(* IEC 61131-3 sources: TIA2AX/tests/V18/test_projects/expected/HW_2200330/ST60_PLC, 7 files *)

(* ---- HwIdentifiers.st ---- *)
TYPE
	HwIdentifiers : WORD
	(
		ST60_PLC_Profilschiene_0 :=	WORD#256,
		ST60_PLC :=	WORD#48,
		ST60_PLC_Card_reader_writer_1 :=	WORD#51,
		ST60_PLC_CPU_display_1 :=	WORD#54,
		ST60_PLC_OPC_UA_1 :=	WORD#117,
		ST60_PLC_DP_interface_1 :=	WORD#60,
		ST60_PLC_PROFINET_interface_1 :=	WORD#64,
		ST60_PLC_PROFINET_interface_1_Port_1 :=	WORD#65,
		ST60_PLC_PROFINET_interface_1_Port_2 :=	WORD#66,
		ST60_PLC_PROFINET_interface_2 :=	WORD#72,
		ST60_PLC_PROFINET_interface_2_Port_1 :=	WORD#73,
		ST60_Switch_SCALANCE_X_rack :=	WORD#421,
		ST60_Switch :=	WORD#422,
		ST60_Switch_ST60_Switch :=	WORD#423,
		ST60_Switch_SCALANCE_interface_1 :=	WORD#424,
		ST60_Switch_SCALANCE_interface_1_Port_1 :=	WORD#425,
		ST60_Switch_SCALANCE_interface_1_Port_2 :=	WORD#426,
		ST60_Switch_SCALANCE_interface_1_Port_3 :=	WORD#427,
		ST60_Switch_SCALANCE_interface_1_Port_4 :=	WORD#428,
		ST60_Switch_SCALANCE_interface_1_Port_5 :=	WORD#429,
		ST60_Switch_SCALANCE_interface_1_Port_6 :=	WORD#430,
		ST60_Switch_SCALANCE_interface_1_Port_7 :=	WORD#431,
		ST60_Switch_SCALANCE_interface_1_Port_8 :=	WORD#432,
		ST60_Switch_SCALANCE_interface_1_Port_9 :=	WORD#433,
		ST60_Switch_SCALANCE_interface_1_Port_10 :=	WORD#434,
		ST60_Switch_SCALANCE_interface_1_Port_11 :=	WORD#435,
		ST60_Switch_SCALANCE_interface_1_Port_12 :=	WORD#436,
		ST60_Switch_SCALANCE_interface_1_Port_13 :=	WORD#437,
		ST60_Switch_SCALANCE_interface_1_Port_14 :=	WORD#438,
		ST60_Switch_SCALANCE_interface_1_Port_15 :=	WORD#439,
		ST60_Switch_SCALANCE_interface_1_Port_16 :=	WORD#440,
		ST60_Switch_1_SCALANCE_X_rack :=	WORD#445,
		ST60_Switch_1 :=	WORD#446,
		ST60_Switch_1_ST60_Switch_1 :=	WORD#447,
		ST60_Switch_1_SCALANCE_interface_1 :=	WORD#448,
		ST60_Switch_1_SCALANCE_interface_1_Port_1 :=	WORD#449,
		ST60_Switch_1_SCALANCE_interface_1_Port_2 :=	WORD#450,
		ST60_Switch_1_SCALANCE_interface_1_Port_3 :=	WORD#451,
		ST60_Switch_1_SCALANCE_interface_1_Port_4 :=	WORD#452,
		ST60_Switch_1_SCALANCE_interface_1_Port_5 :=	WORD#453,
		ST60_Switch_1_SCALANCE_interface_1_Port_6 :=	WORD#454,
		ST60_Switch_1_SCALANCE_interface_1_Port_7 :=	WORD#455,
		ST60_Switch_1_SCALANCE_interface_1_Port_8 :=	WORD#456,
		ST60_Switch_1_SCALANCE_interface_1_Port_9 :=	WORD#457,
		ST60_Switch_1_SCALANCE_interface_1_Port_10 :=	WORD#458,
		ST60_Switch_1_SCALANCE_interface_1_Port_11 :=	WORD#459,
		ST60_Switch_1_SCALANCE_interface_1_Port_12 :=	WORD#460,
		ST60_Switch_1_SCALANCE_interface_1_Port_13 :=	WORD#461,
		ST60_Switch_1_SCALANCE_interface_1_Port_14 :=	WORD#462,
		ST60_Switch_1_SCALANCE_interface_1_Port_15 :=	WORD#463,
		ST60_Switch_1_SCALANCE_interface_1_Port_16 :=	WORD#464,
		ST60_2_DM260_Rack :=	WORD#270,
		ST60_2_DM260 :=	WORD#258,
		ST60_2_DM260_Interface :=	WORD#259,
		ST60_2_DM260_Interface_Port_1 :=	WORD#260,
		ST60_2_DM260_DataMan_260 :=	WORD#261,
		ST60_2_DM260_Acquisition_Control :=	WORD#262,
		ST60_2_DM260_Acquisition_Status :=	WORD#263,
		ST60_2_DM260_Results_Control :=	WORD#264,
		ST60_2_DM260_Results_Status :=	WORD#265,
		ST60_2_DM260_Soft_Event_Control :=	WORD#266,
		ST60_2_DM260_User_Data_64_bytes :=	WORD#267,
		ST60_2_DM260_Result_Data_64_bytes :=	WORD#268,
		ST60_1_DM260_Rack :=	WORD#272,
		ST60_1_DM260 :=	WORD#273,
		ST60_1_DM260_Interface :=	WORD#274,
		ST60_1_DM260_Interface_Port_1 :=	WORD#275,
		ST60_1_DM260_DataMan_260 :=	WORD#276,
		ST60_1_DM260_Acquisition_Control :=	WORD#277,
		ST60_1_DM260_Acquisition_Status :=	WORD#278,
		ST60_1_DM260_Results_Control :=	WORD#279,
		ST60_1_DM260_Results_Status :=	WORD#280,
		ST60_1_DM260_Soft_Event_Control :=	WORD#281,
		ST60_1_DM260_User_Data_64_bytes :=	WORD#282,
		ST60_1_DM260_Result_Data_64_bytes :=	WORD#283,
		ST60_1_DM260_WPC_Rack :=	WORD#285,
		ST60_1_DM260_WPC :=	WORD#286,
		ST60_1_DM260_WPC_Interface :=	WORD#287,
		ST60_1_DM260_WPC_Interface_Port_1 :=	WORD#288,
		ST60_1_DM260_WPC_DataMan_260 :=	WORD#289,
		ST60_1_DM260_WPC_Acquisition_Control :=	WORD#290,
		ST60_1_DM260_WPC_Acquisition_Status :=	WORD#291,
		ST60_1_DM260_WPC_Results_Control :=	WORD#292,
		ST60_1_DM260_WPC_Results_Status :=	WORD#293,
		ST60_1_DM260_WPC_Soft_Event_Control :=	WORD#294,
		ST60_1_DM260_WPC_User_Data_64_bytes :=	WORD#295,
		ST60_1_DM260_WPC_Result_Data_64_bytes :=	WORD#296,
		ST60_TZ535_PN_Rack :=	WORD#298,
		ST60_TZ535_PN :=	WORD#299,
		ST60_TZ535_PN_Interface :=	WORD#300,
		ST60_TZ535_PN_Interface_Port_1 :=	WORD#301,
		ST60_TZ535_PN_Interface_Port_2 :=	WORD#302,
		ST60_TZ535_PN_2D_TZ535_PN_PROFINET_IO :=	WORD#303,
		ST60_TZ535_PN_In_Out_32_byte_x :=	WORD#304,
		ST60_SCHUNK_R_Rack :=	WORD#306,
		ST60_SCHUNK_R :=	WORD#307,
		ST60_SCHUNK_R_Interface :=	WORD#308,
		ST60_SCHUNK_R_Interface_Port_1 :=	WORD#309,
		ST60_SCHUNK_R_Interface_Port_2 :=	WORD#310,
		ST60_SCHUNK_R_DEVICE_SFP :=	WORD#311,
		ST60_SCHUNK_R_IN_4_Double_Words :=	WORD#312,
		ST60_SCHUNK_R_OUT_4_Double_Words :=	WORD#313,
		ST60_SCHUNK_L_Rack :=	WORD#315,
		ST60_SCHUNK_L :=	WORD#316,
		ST60_SCHUNK_L_Interface :=	WORD#317,
		ST60_SCHUNK_L_Interface_Port_1 :=	WORD#318,
		ST60_SCHUNK_L_Interface_Port_2 :=	WORD#319,
		ST60_SCHUNK_L_DEVICE_SFP :=	WORD#320,
		ST60_SCHUNK_L_IN_4_Double_Words :=	WORD#321,
		ST60_SCHUNK_L_OUT_4_Double_Words :=	WORD#322,
		ST60_CPX_PN_IO_Interface :=	WORD#326,
		ST60_CPX_PN_IO_Interface_Port_1 :=	WORD#327,
		ST60_CPX_PN_IO_Interface_Port_2 :=	WORD#328,
		ST60_CPX_CPX :=	WORD#329,
		ST60_CPX_MPA1S_VMPA1_FB_EMS_8_8DO_1 :=	WORD#330,
		ST60_CPX_MPA1S_VMPA1_FB_EMS_8_8DO_2 :=	WORD#331,
		ST60_CPX_MPA1S_VMPA1_FB_EMS_8_8DO_3 :=	WORD#332,
		ST60_CPX_MPA1S_VMPA1_FB_EMS_8_8DO_4 :=	WORD#333,
		ST60_CPX_MPA1S_VMPA1_FB_EMS_8_8DO_5 :=	WORD#334,
		ST60_CPX_MPA1S_VMPA1_FB_EMS_8_8DO_6 :=	WORD#335,
		ST60_CPX_MPA1S_VMPA1_FB_EMS_8_8DO_7 :=	WORD#336,
		ST60_CPX_MPA1S_VMPA1_FB_EMS_8_8DO_8 :=	WORD#337,
		ST60_CPX_MPA1S_VMPA1_FB_EMS_8_8DO_9 :=	WORD#338,
		ST60_CPX_MPA1G_VMPA1_FB_EMG_8_8DO_4 :=	WORD#339,
		ST60_ET200SP_Rack_0 :=	WORD#341,
		ST60_ET200SP :=	WORD#342,
		ST60_ET200SP_ST60_ET200SP :=	WORD#343,
		ST60_ET200SP_PROFINET_interface :=	WORD#344,
		ST60_ET200SP_PROFINET_interface_Port_1 :=	WORD#346,
		ST60_ET200SP_PROFINET_interface_Port_2 :=	WORD#345,
		ST60_ET200SP_BA_2xRJ45 :=	WORD#346,
		ST60_ET200SP_CM_4xIO_Link_1 :=	WORD#347,
		ST60_ET200SP_CM_4xIO_Link_2 :=	WORD#348,
		ST60_ET200SP_CM_4xIO_Link_3 :=	WORD#349,
		ST60_ET200SP_AI_4xI_2_4_wire_ST_1 :=	WORD#350,
		ST60_ET200SP_DI_16x24VDC_ST_1 :=	WORD#351,
		ST60_ET200SP_DI_16x24VDC_ST_2 :=	WORD#352,
		ST60_ET200SP_DI_8x24VDC_ST_4 :=	WORD#353,
		ST60_ET200SP_DI_8x24VDC_ST_3 :=	WORD#354,
		ST60_ET200SP_DQ_16x24VDC_0_5A_ST_1 :=	WORD#355,
		ST60_ET200SP_DQ_16x24VDC_0_5A_ST_2 :=	WORD#356,
		ST60_ET200SP_DQ_16x24VDC_0_5A_ST_3 :=	WORD#357,
		ST60_ET200SP_DQ_16x24VDC_0_5A_ST_4 :=	WORD#358,
		ST60_ET200SP_Servermodul_1 :=	WORD#359,
		ST60_HMI_ConnectionBox_Connection_Box :=	WORD#361,
		ST60_HMI_ConnectionBox :=	WORD#362,
		ST60_HMI_ConnectionBox_ST60_HMI_ConnectionBox :=	WORD#363,
		ST60_HMI_ConnectionBox_SCALANCE_interface_1 :=	WORD#364,
		ST60_HMI_ConnectionBox_SCALANCE_interface_1_Port_1 :=	WORD#365,
		ST60_HMI_ConnectionBox_SCALANCE_interface_1_Port_2 :=	WORD#366,
		ST60_HMI_ConnectionBox_SCALANCE_interface_1_Port_3 :=	WORD#367,
		ST60_6_DM260_Rack :=	WORD#369,
		ST60_6_DM260 :=	WORD#370,
		ST60_6_DM260_Interface :=	WORD#371,
		ST60_6_DM260_Interface_Port_1 :=	WORD#372,
		ST60_6_DM260_DataMan_260 :=	WORD#373,
		ST60_6_DM260_Acquisition_Control :=	WORD#374,
		ST60_6_DM260_Acquisition_Status :=	WORD#375,
		ST60_6_DM260_Results_Control :=	WORD#376,
		ST60_6_DM260_Results_Status :=	WORD#377,
		ST60_6_DM260_Soft_Event_Control :=	WORD#378,
		ST60_6_DM260_User_Data_64_bytes :=	WORD#379,
		ST60_6_DM260_Result_Data_64_bytes :=	WORD#380,
		ST60_3_DM260_Rack :=	WORD#382,
		ST60_3_DM260 :=	WORD#383,
		ST60_3_DM260_Interface :=	WORD#384,
		ST60_3_DM260_Interface_Port_1 :=	WORD#385,
		ST60_3_DM260_DataMan_260 :=	WORD#386,
		ST60_3_DM260_Acquisition_Control :=	WORD#387,
		ST60_3_DM260_Acquisition_Status :=	WORD#388,
		ST60_3_DM260_Results_Control :=	WORD#389,
		ST60_3_DM260_Results_Status :=	WORD#390,
		ST60_3_DM260_Soft_Event_Control :=	WORD#391,
		ST60_3_DM260_User_Data_64_bytes :=	WORD#392,
		ST60_3_DM260_Result_Data_64_bytes :=	WORD#393,
		ST60_4_DM260_Rack :=	WORD#395,
		ST60_4_DM260 :=	WORD#396,
		ST60_4_DM260_Interface :=	WORD#397,
		ST60_4_DM260_Interface_Port_1 :=	WORD#398,
		ST60_4_DM260_DataMan_260 :=	WORD#399,
		ST60_4_DM260_Acquisition_Control :=	WORD#400,
		ST60_4_DM260_Acquisition_Status :=	WORD#401,
		ST60_4_DM260_Results_Control :=	WORD#402,
		ST60_4_DM260_Results_Status :=	WORD#403,
		ST60_4_DM260_Soft_Event_Control :=	WORD#404,
		ST60_4_DM260_User_Data_64_bytes :=	WORD#405,
		ST60_4_DM260_Result_Data_64_bytes :=	WORD#406,
		ST60_5_DM260_Rack :=	WORD#408,
		ST60_5_DM260 :=	WORD#409,
		ST60_5_DM260_Interface :=	WORD#410,
		ST60_5_DM260_Interface_Port_1 :=	WORD#411,
		ST60_5_DM260_DataMan_260 :=	WORD#412,
		ST60_5_DM260_Acquisition_Control :=	WORD#413,
		ST60_5_DM260_Acquisition_Status :=	WORD#414,
		ST60_5_DM260_Results_Control :=	WORD#415,
		ST60_5_DM260_Results_Status :=	WORD#416,
		ST60_5_DM260_Soft_Event_Control :=	WORD#417,
		ST60_5_DM260_User_Data_64_bytes :=	WORD#418,
		ST60_5_DM260_Result_Data_64_bytes :=	WORD#419,
		NONE:= WORD#0
	);
END_TYPE

(* ---- HwInputs.st ---- *)
TYPE
	HwInputs : STRUCT
		ST60_2_DM260_Acquisition_Status AT %B3731 : ARRAY[0..2] OF BYTE;
		ST60_2_DM260_Results_Status AT %B3734 : BYTE;
		ST60_2_DM260_Soft_Event_Control AT %B3735 : BYTE;
		ST60_2_DM260_Result_Data_64_bytes AT %B3736 : ARRAY[0..71] OF BYTE;
		ST60_1_DM260_Acquisition_Status AT %B3654 : ARRAY[0..2] OF BYTE;
		ST60_1_DM260_Results_Status AT %B3657 : BYTE;
		ST60_1_DM260_Soft_Event_Control AT %B3658 : BYTE;
		ST60_1_DM260_Result_Data_64_bytes AT %B3659 : ARRAY[0..71] OF BYTE;
		ST60_1_DM260_WPC_Acquisition_Status AT %B3500 : ARRAY[0..2] OF BYTE;
		ST60_1_DM260_WPC_Results_Status AT %B3503 : BYTE;
		ST60_1_DM260_WPC_Soft_Event_Control AT %B3504 : BYTE;
		ST60_1_DM260_WPC_Result_Data_64_bytes AT %B3510 : ARRAY[0..71] OF BYTE;
		ST60_TZ535_PN_In_Out_32_byte_x AT %B1000 : ARRAY[0..31] OF BYTE;
		ST60_SCHUNK_R_IN_4_Double_Words AT %B616 : ARRAY[0..15] OF BYTE;
		ST60_SCHUNK_L_IN_4_Double_Words AT %B600 : ARRAY[0..15] OF BYTE;
		ST60_ET200SP_CM_4xIO_Link_1 AT %B100 : ARRAY[0..31] OF BYTE;
		ST60_ET200SP_CM_4xIO_Link_2 AT %B132 : ARRAY[0..31] OF BYTE;
		ST60_ET200SP_CM_4xIO_Link_3 AT %B164 : ARRAY[0..31] OF BYTE;
		ST60_ET200SP_AI_4xI_2_4_wire_ST_1 AT %B6 : ARRAY[0..7] OF BYTE;
		ST60_ET200SP_DI_16x24VDC_ST_1 AT %B0 : WORD;
		ST60_ET200SP_DI_16x24VDC_ST_2 AT %B2 : WORD;
		ST60_ET200SP_DI_8x24VDC_ST_4 AT %B4 : BYTE;
		ST60_ET200SP_DI_8x24VDC_ST_3 AT %B5 : BYTE;
		ST60_6_DM260_Acquisition_Status AT %B9100 : ARRAY[0..2] OF BYTE;
		ST60_6_DM260_Results_Status AT %B9103 : BYTE;
		ST60_6_DM260_Soft_Event_Control AT %B9104 : BYTE;
		ST60_6_DM260_Result_Data_64_bytes AT %B9110 : ARRAY[0..71] OF BYTE;
		ST60_3_DM260_Acquisition_Status AT %B3808 : ARRAY[0..2] OF BYTE;
		ST60_3_DM260_Results_Status AT %B3811 : BYTE;
		ST60_3_DM260_Soft_Event_Control AT %B3812 : BYTE;
		ST60_3_DM260_Result_Data_64_bytes AT %B3813 : ARRAY[0..71] OF BYTE;
		ST60_4_DM260_Acquisition_Status AT %B3885 : ARRAY[0..2] OF BYTE;
		ST60_4_DM260_Results_Status AT %B3888 : BYTE;
		ST60_4_DM260_Soft_Event_Control AT %B3889 : BYTE;
		ST60_4_DM260_Result_Data_64_bytes AT %B3890 : ARRAY[0..71] OF BYTE;
		ST60_5_DM260_Acquisition_Status AT %B3962 : ARRAY[0..2] OF BYTE;
		ST60_5_DM260_Results_Status AT %B3965 : BYTE;
		ST60_5_DM260_Soft_Event_Control AT %B3966 : BYTE;
		ST60_5_DM260_Result_Data_64_bytes AT %B3967 : ARRAY[0..71] OF BYTE;
	END_STRUCT;
END_TYPE

(* ---- HwOutputs.st ---- *)
TYPE
	HwOutputs : STRUCT
		ST60_2_DM260_Acquisition_Control AT %B3509 : BYTE;
		ST60_2_DM260_Results_Control AT %B3714 : BYTE;
		ST60_2_DM260_Soft_Event_Control AT %B3715 : BYTE;
		ST60_2_DM260_User_Data_64_bytes AT %B3716 : ARRAY[0..67] OF BYTE;
		ST60_1_DM260_Acquisition_Control AT %B3502 : BYTE;
		ST60_1_DM260_Results_Control AT %B3507 : BYTE;
		ST60_1_DM260_Soft_Event_Control AT %B3508 : BYTE;
		ST60_1_DM260_User_Data_64_bytes AT %B3646 : ARRAY[0..67] OF BYTE;
		ST60_1_DM260_WPC_Acquisition_Control AT %B3500 : BYTE;
		ST60_1_DM260_WPC_Results_Control AT %B3503 : BYTE;
		ST60_1_DM260_WPC_Soft_Event_Control AT %B3504 : BYTE;
		ST60_1_DM260_WPC_User_Data_64_bytes AT %B3510 : ARRAY[0..67] OF BYTE;
		ST60_TZ535_PN_In_Out_32_byte_x AT %B1000 : ARRAY[0..31] OF BYTE;
		ST60_SCHUNK_R_OUT_4_Double_Words AT %B616 : ARRAY[0..15] OF BYTE;
		ST60_SCHUNK_L_OUT_4_Double_Words AT %B600 : ARRAY[0..15] OF BYTE;
		ST60_CPX_MPA1S_VMPA1_FB_EMS_8_8DO_1 AT %B200 : BYTE;
		ST60_CPX_MPA1S_VMPA1_FB_EMS_8_8DO_2 AT %B201 : BYTE;
		ST60_CPX_MPA1S_VMPA1_FB_EMS_8_8DO_3 AT %B202 : BYTE;
		ST60_CPX_MPA1S_VMPA1_FB_EMS_8_8DO_4 AT %B203 : BYTE;
		ST60_CPX_MPA1S_VMPA1_FB_EMS_8_8DO_5 AT %B204 : BYTE;
		ST60_CPX_MPA1S_VMPA1_FB_EMS_8_8DO_6 AT %B205 : BYTE;
		ST60_CPX_MPA1S_VMPA1_FB_EMS_8_8DO_7 AT %B206 : BYTE;
		ST60_CPX_MPA1S_VMPA1_FB_EMS_8_8DO_8 AT %B207 : BYTE;
		ST60_CPX_MPA1S_VMPA1_FB_EMS_8_8DO_9 AT %B208 : BYTE;
		ST60_CPX_MPA1G_VMPA1_FB_EMG_8_8DO_4 AT %B209 : BYTE;
		ST60_ET200SP_CM_4xIO_Link_1 AT %B100 : ARRAY[0..31] OF BYTE;
		ST60_ET200SP_CM_4xIO_Link_2 AT %B132 : ARRAY[0..31] OF BYTE;
		ST60_ET200SP_CM_4xIO_Link_3 AT %B164 : ARRAY[0..31] OF BYTE;
		ST60_ET200SP_DQ_16x24VDC_0_5A_ST_1 AT %B0 : WORD;
		ST60_ET200SP_DQ_16x24VDC_0_5A_ST_2 AT %B2 : WORD;
		ST60_ET200SP_DQ_16x24VDC_0_5A_ST_3 AT %B4 : WORD;
		ST60_ET200SP_DQ_16x24VDC_0_5A_ST_4 AT %B6 : WORD;
		ST60_6_DM260_Acquisition_Control AT %B9100 : BYTE;
		ST60_6_DM260_Results_Control AT %B9103 : BYTE;
		ST60_6_DM260_Soft_Event_Control AT %B9104 : BYTE;
		ST60_6_DM260_User_Data_64_bytes AT %B9110 : ARRAY[0..67] OF BYTE;
		ST60_3_DM260_Acquisition_Control AT %B3784 : BYTE;
		ST60_3_DM260_Results_Control AT %B3785 : BYTE;
		ST60_3_DM260_Soft_Event_Control AT %B3786 : BYTE;
		ST60_3_DM260_User_Data_64_bytes AT %B3787 : ARRAY[0..67] OF BYTE;
		ST60_4_DM260_Acquisition_Control AT %B3855 : BYTE;
		ST60_4_DM260_Results_Control AT %B3856 : BYTE;
		ST60_4_DM260_Soft_Event_Control AT %B3857 : BYTE;
		ST60_4_DM260_User_Data_64_bytes AT %B3858 : ARRAY[0..67] OF BYTE;
		ST60_5_DM260_Acquisition_Control AT %B3926 : BYTE;
		ST60_5_DM260_Results_Control AT %B3927 : BYTE;
		ST60_5_DM260_Soft_Event_Control AT %B3928 : BYTE;
		ST60_5_DM260_User_Data_64_bytes AT %B3929 : ARRAY[0..67] OF BYTE;
	END_STRUCT;
END_TYPE

(* ---- PlcInputs.st ---- *)
TYPE
	PlcInputs : STRUCT
		ST60_2_DM260_Acquisition_Status : ARRAY[0..2] OF BYTE;
		ST60_2_DM260_Results_Status : BYTE;
		ST60_2_DM260_Soft_Event_Control : BYTE;
		ST60_2_DM260_Result_Data_64_bytes : ARRAY[0..71] OF BYTE;
		ST60_1_DM260_Acquisition_Status : ARRAY[0..2] OF BYTE;
		ST60_1_DM260_Results_Status : BYTE;
		ST60_1_DM260_Soft_Event_Control : BYTE;
		ST60_1_DM260_Result_Data_64_bytes : ARRAY[0..71] OF BYTE;
		ST60_1_DM260_WPC_Acquisition_Status : ARRAY[0..2] OF BYTE;
		ST60_1_DM260_WPC_Results_Status : BYTE;
		ST60_1_DM260_WPC_Soft_Event_Control : BYTE;
		ST60_1_DM260_WPC_Result_Data_64_bytes : ARRAY[0..71] OF BYTE;
		ST60_TZ535_PN_In_Out_32_byte_x : ARRAY[0..31] OF BYTE;
		ST60_SCHUNK_R_IN_4_Double_Words : ARRAY[0..15] OF BYTE;
		ST60_SCHUNK_L_IN_4_Double_Words : ARRAY[0..15] OF BYTE;
		ST60_ET200SP_CM_4xIO_Link_1 : ARRAY[0..31] OF BYTE;
		ST60_ET200SP_CM_4xIO_Link_2 : ARRAY[0..31] OF BYTE;
		ST60_ET200SP_CM_4xIO_Link_3 : ARRAY[0..31] OF BYTE;
		ST60_ET200SP_AI_4xI_2_4_wire_ST_1 : ARRAY[0..7] OF BYTE;
		ST60_ET200SP_DI_16x24VDC_ST_1 : WORD;
		ST60_ET200SP_DI_16x24VDC_ST_2 : WORD;
		ST60_ET200SP_DI_8x24VDC_ST_4 : BYTE;
		ST60_ET200SP_DI_8x24VDC_ST_3 : BYTE;
		ST60_6_DM260_Acquisition_Status : ARRAY[0..2] OF BYTE;
		ST60_6_DM260_Results_Status : BYTE;
		ST60_6_DM260_Soft_Event_Control : BYTE;
		ST60_6_DM260_Result_Data_64_bytes : ARRAY[0..71] OF BYTE;
		ST60_3_DM260_Acquisition_Status : ARRAY[0..2] OF BYTE;
		ST60_3_DM260_Results_Status : BYTE;
		ST60_3_DM260_Soft_Event_Control : BYTE;
		ST60_3_DM260_Result_Data_64_bytes : ARRAY[0..71] OF BYTE;
		ST60_4_DM260_Acquisition_Status : ARRAY[0..2] OF BYTE;
		ST60_4_DM260_Results_Status : BYTE;
		ST60_4_DM260_Soft_Event_Control : BYTE;
		ST60_4_DM260_Result_Data_64_bytes : ARRAY[0..71] OF BYTE;
		ST60_5_DM260_Acquisition_Status : ARRAY[0..2] OF BYTE;
		ST60_5_DM260_Results_Status : BYTE;
		ST60_5_DM260_Soft_Event_Control : BYTE;
		ST60_5_DM260_Result_Data_64_bytes : ARRAY[0..71] OF BYTE;
	END_STRUCT;
END_TYPE

(* ---- PlcOutputs.st ---- *)
TYPE
	PlcOutputs : STRUCT
		ST60_2_DM260_Acquisition_Control : BYTE;
		ST60_2_DM260_Results_Control : BYTE;
		ST60_2_DM260_Soft_Event_Control : BYTE;
		ST60_2_DM260_User_Data_64_bytes : ARRAY[0..67] OF BYTE;
		ST60_1_DM260_Acquisition_Control : BYTE;
		ST60_1_DM260_Results_Control : BYTE;
		ST60_1_DM260_Soft_Event_Control : BYTE;
		ST60_1_DM260_User_Data_64_bytes : ARRAY[0..67] OF BYTE;
		ST60_1_DM260_WPC_Acquisition_Control : BYTE;
		ST60_1_DM260_WPC_Results_Control : BYTE;
		ST60_1_DM260_WPC_Soft_Event_Control : BYTE;
		ST60_1_DM260_WPC_User_Data_64_bytes : ARRAY[0..67] OF BYTE;
		ST60_TZ535_PN_In_Out_32_byte_x : ARRAY[0..31] OF BYTE;
		ST60_SCHUNK_R_OUT_4_Double_Words : ARRAY[0..15] OF BYTE;
		ST60_SCHUNK_L_OUT_4_Double_Words : ARRAY[0..15] OF BYTE;
		ST60_CPX_MPA1S_VMPA1_FB_EMS_8_8DO_1 : BYTE;
		ST60_CPX_MPA1S_VMPA1_FB_EMS_8_8DO_2 : BYTE;
		ST60_CPX_MPA1S_VMPA1_FB_EMS_8_8DO_3 : BYTE;
		ST60_CPX_MPA1S_VMPA1_FB_EMS_8_8DO_4 : BYTE;
		ST60_CPX_MPA1S_VMPA1_FB_EMS_8_8DO_5 : BYTE;
		ST60_CPX_MPA1S_VMPA1_FB_EMS_8_8DO_6 : BYTE;
		ST60_CPX_MPA1S_VMPA1_FB_EMS_8_8DO_7 : BYTE;
		ST60_CPX_MPA1S_VMPA1_FB_EMS_8_8DO_8 : BYTE;
		ST60_CPX_MPA1S_VMPA1_FB_EMS_8_8DO_9 : BYTE;
		ST60_CPX_MPA1G_VMPA1_FB_EMG_8_8DO_4 : BYTE;
		ST60_ET200SP_CM_4xIO_Link_1 : ARRAY[0..31] OF BYTE;
		ST60_ET200SP_CM_4xIO_Link_2 : ARRAY[0..31] OF BYTE;
		ST60_ET200SP_CM_4xIO_Link_3 : ARRAY[0..31] OF BYTE;
		ST60_ET200SP_DQ_16x24VDC_0_5A_ST_1 : WORD;
		ST60_ET200SP_DQ_16x24VDC_0_5A_ST_2 : WORD;
		ST60_ET200SP_DQ_16x24VDC_0_5A_ST_3 : WORD;
		ST60_ET200SP_DQ_16x24VDC_0_5A_ST_4 : WORD;
		ST60_6_DM260_Acquisition_Control : BYTE;
		ST60_6_DM260_Results_Control : BYTE;
		ST60_6_DM260_Soft_Event_Control : BYTE;
		ST60_6_DM260_User_Data_64_bytes : ARRAY[0..67] OF BYTE;
		ST60_3_DM260_Acquisition_Control : BYTE;
		ST60_3_DM260_Results_Control : BYTE;
		ST60_3_DM260_Soft_Event_Control : BYTE;
		ST60_3_DM260_User_Data_64_bytes : ARRAY[0..67] OF BYTE;
		ST60_4_DM260_Acquisition_Control : BYTE;
		ST60_4_DM260_Results_Control : BYTE;
		ST60_4_DM260_Soft_Event_Control : BYTE;
		ST60_4_DM260_User_Data_64_bytes : ARRAY[0..67] OF BYTE;
		ST60_5_DM260_Acquisition_Control : BYTE;
		ST60_5_DM260_Results_Control : BYTE;
		ST60_5_DM260_Soft_Event_Control : BYTE;
		ST60_5_DM260_User_Data_64_bytes : ARRAY[0..67] OF BYTE;
	END_STRUCT;
END_TYPE

(* ---- CopyInputs.st ---- *)
FUNCTION CopyInputs
	VAR_EXTERNAL
		HwInputs : HwInputs;
		PlcInputs : PlcInputs;
	END_VAR
	PlcInputs.ST60_2_DM260_Acquisition_Status[0] := HwInputs.ST60_2_DM260_Acquisition_Status[0];
	PlcInputs.ST60_2_DM260_Acquisition_Status[1] := HwInputs.ST60_2_DM260_Acquisition_Status[1];
	PlcInputs.ST60_2_DM260_Acquisition_Status[2] := HwInputs.ST60_2_DM260_Acquisition_Status[2];
	PlcInputs.ST60_2_DM260_Results_Status := HwInputs.ST60_2_DM260_Results_Status;
	PlcInputs.ST60_2_DM260_Soft_Event_Control := HwInputs.ST60_2_DM260_Soft_Event_Control;
	PlcInputs.ST60_2_DM260_Result_Data_64_bytes[0] := HwInputs.ST60_2_DM260_Result_Data_64_bytes[0];
	PlcInputs.ST60_2_DM260_Result_Data_64_bytes[1] := HwInputs.ST60_2_DM260_Result_Data_64_bytes[1];
	PlcInputs.ST60_2_DM260_Result_Data_64_bytes[2] := HwInputs.ST60_2_DM260_Result_Data_64_bytes[2];
	PlcInputs.ST60_2_DM260_Result_Data_64_bytes[3] := HwInputs.ST60_2_DM260_Result_Data_64_bytes[3];
	PlcInputs.ST60_2_DM260_Result_Data_64_bytes[4] := HwInputs.ST60_2_DM260_Result_Data_64_bytes[4];
	PlcInputs.ST60_2_DM260_Result_Data_64_bytes[5] := HwInputs.ST60_2_DM260_Result_Data_64_bytes[5];
	PlcInputs.ST60_2_DM260_Result_Data_64_bytes[6] := HwInputs.ST60_2_DM260_Result_Data_64_bytes[6];
	PlcInputs.ST60_2_DM260_Result_Data_64_bytes[7] := HwInputs.ST60_2_DM260_Result_Data_64_bytes[7];
	PlcInputs.ST60_2_DM260_Result_Data_64_bytes[8] := HwInputs.ST60_2_DM260_Result_Data_64_bytes[8];
	PlcInputs.ST60_2_DM260_Result_Data_64_bytes[9] := HwInputs.ST60_2_DM260_Result_Data_64_bytes[9];
	PlcInputs.ST60_2_DM260_Result_Data_64_bytes[10] := HwInputs.ST60_2_DM260_Result_Data_64_bytes[10];
	PlcInputs.ST60_2_DM260_Result_Data_64_bytes[11] := HwInputs.ST60_2_DM260_Result_Data_64_bytes[11];
	PlcInputs.ST60_2_DM260_Result_Data_64_bytes[12] := HwInputs.ST60_2_DM260_Result_Data_64_bytes[12];
	PlcInputs.ST60_2_DM260_Result_Data_64_bytes[13] := HwInputs.ST60_2_DM260_Result_Data_64_bytes[13];
	PlcInputs.ST60_2_DM260_Result_Data_64_bytes[14] := HwInputs.ST60_2_DM260_Result_Data_64_bytes[14];
	PlcInputs.ST60_2_DM260_Result_Data_64_bytes[15] := HwInputs.ST60_2_DM260_Result_Data_64_bytes[15];
	PlcInputs.ST60_2_DM260_Result_Data_64_bytes[16] := HwInputs.ST60_2_DM260_Result_Data_64_bytes[16];
	PlcInputs.ST60_2_DM260_Result_Data_64_bytes[17] := HwInputs.ST60_2_DM260_Result_Data_64_bytes[17];
	PlcInputs.ST60_2_DM260_Result_Data_64_bytes[18] := HwInputs.ST60_2_DM260_Result_Data_64_bytes[18];
	PlcInputs.ST60_2_DM260_Result_Data_64_bytes[19] := HwInputs.ST60_2_DM260_Result_Data_64_bytes[19];
	PlcInputs.ST60_2_DM260_Result_Data_64_bytes[20] := HwInputs.ST60_2_DM260_Result_Data_64_bytes[20];
	PlcInputs.ST60_2_DM260_Result_Data_64_bytes[21] := HwInputs.ST60_2_DM260_Result_Data_64_bytes[21];
	PlcInputs.ST60_2_DM260_Result_Data_64_bytes[22] := HwInputs.ST60_2_DM260_Result_Data_64_bytes[22];
	PlcInputs.ST60_2_DM260_Result_Data_64_bytes[23] := HwInputs.ST60_2_DM260_Result_Data_64_bytes[23];
	PlcInputs.ST60_2_DM260_Result_Data_64_bytes[24] := HwInputs.ST60_2_DM260_Result_Data_64_bytes[24];
	PlcInputs.ST60_2_DM260_Result_Data_64_bytes[25] := HwInputs.ST60_2_DM260_Result_Data_64_bytes[25];
	PlcInputs.ST60_2_DM260_Result_Data_64_bytes[26] := HwInputs.ST60_2_DM260_Result_Data_64_bytes[26];
	PlcInputs.ST60_2_DM260_Result_Data_64_bytes[27] := HwInputs.ST60_2_DM260_Result_Data_64_bytes[27];
	PlcInputs.ST60_2_DM260_Result_Data_64_bytes[28] := HwInputs.ST60_2_DM260_Result_Data_64_bytes[28];
	PlcInputs.ST60_2_DM260_Result_Data_64_bytes[29] := HwInputs.ST60_2_DM260_Result_Data_64_bytes[29];
	PlcInputs.ST60_2_DM260_Result_Data_64_bytes[30] := HwInputs.ST60_2_DM260_Result_Data_64_bytes[30];
	PlcInputs.ST60_2_DM260_Result_Data_64_bytes[31] := HwInputs.ST60_2_DM260_Result_Data_64_bytes[31];
	PlcInputs.ST60_2_DM260_Result_Data_64_bytes[32] := HwInputs.ST60_2_DM260_Result_Data_64_bytes[32];
	PlcInputs.ST60_2_DM260_Result_Data_64_bytes[33] := HwInputs.ST60_2_DM260_Result_Data_64_bytes[33];
	PlcInputs.ST60_2_DM260_Result_Data_64_bytes[34] := HwInputs.ST60_2_DM260_Result_Data_64_bytes[34];
	PlcInputs.ST60_2_DM260_Result_Data_64_bytes[35] := HwInputs.ST60_2_DM260_Result_Data_64_bytes[35];
	PlcInputs.ST60_2_DM260_Result_Data_64_bytes[36] := HwInputs.ST60_2_DM260_Result_Data_64_bytes[36];
	PlcInputs.ST60_2_DM260_Result_Data_64_bytes[37] := HwInputs.ST60_2_DM260_Result_Data_64_bytes[37];
	PlcInputs.ST60_2_DM260_Result_Data_64_bytes[38] := HwInputs.ST60_2_DM260_Result_Data_64_bytes[38];
	PlcInputs.ST60_2_DM260_Result_Data_64_bytes[39] := HwInputs.ST60_2_DM260_Result_Data_64_bytes[39];
	PlcInputs.ST60_2_DM260_Result_Data_64_bytes[40] := HwInputs.ST60_2_DM260_Result_Data_64_bytes[40];
	PlcInputs.ST60_2_DM260_Result_Data_64_bytes[41] := HwInputs.ST60_2_DM260_Result_Data_64_bytes[41];
	PlcInputs.ST60_2_DM260_Result_Data_64_bytes[42] := HwInputs.ST60_2_DM260_Result_Data_64_bytes[42];
	PlcInputs.ST60_2_DM260_Result_Data_64_bytes[43] := HwInputs.ST60_2_DM260_Result_Data_64_bytes[43];
	PlcInputs.ST60_2_DM260_Result_Data_64_bytes[44] := HwInputs.ST60_2_DM260_Result_Data_64_bytes[44];
	PlcInputs.ST60_2_DM260_Result_Data_64_bytes[45] := HwInputs.ST60_2_DM260_Result_Data_64_bytes[45];
	PlcInputs.ST60_2_DM260_Result_Data_64_bytes[46] := HwInputs.ST60_2_DM260_Result_Data_64_bytes[46];
	PlcInputs.ST60_2_DM260_Result_Data_64_bytes[47] := HwInputs.ST60_2_DM260_Result_Data_64_bytes[47];
	PlcInputs.ST60_2_DM260_Result_Data_64_bytes[48] := HwInputs.ST60_2_DM260_Result_Data_64_bytes[48];
	PlcInputs.ST60_2_DM260_Result_Data_64_bytes[49] := HwInputs.ST60_2_DM260_Result_Data_64_bytes[49];
	PlcInputs.ST60_2_DM260_Result_Data_64_bytes[50] := HwInputs.ST60_2_DM260_Result_Data_64_bytes[50];
	PlcInputs.ST60_2_DM260_Result_Data_64_bytes[51] := HwInputs.ST60_2_DM260_Result_Data_64_bytes[51];
	PlcInputs.ST60_2_DM260_Result_Data_64_bytes[52] := HwInputs.ST60_2_DM260_Result_Data_64_bytes[52];
	PlcInputs.ST60_2_DM260_Result_Data_64_bytes[53] := HwInputs.ST60_2_DM260_Result_Data_64_bytes[53];
	PlcInputs.ST60_2_DM260_Result_Data_64_bytes[54] := HwInputs.ST60_2_DM260_Result_Data_64_bytes[54];
	PlcInputs.ST60_2_DM260_Result_Data_64_bytes[55] := HwInputs.ST60_2_DM260_Result_Data_64_bytes[55];
	PlcInputs.ST60_2_DM260_Result_Data_64_bytes[56] := HwInputs.ST60_2_DM260_Result_Data_64_bytes[56];
	PlcInputs.ST60_2_DM260_Result_Data_64_bytes[57] := HwInputs.ST60_2_DM260_Result_Data_64_bytes[57];
	PlcInputs.ST60_2_DM260_Result_Data_64_bytes[58] := HwInputs.ST60_2_DM260_Result_Data_64_bytes[58];
	PlcInputs.ST60_2_DM260_Result_Data_64_bytes[59] := HwInputs.ST60_2_DM260_Result_Data_64_bytes[59];
	PlcInputs.ST60_2_DM260_Result_Data_64_bytes[60] := HwInputs.ST60_2_DM260_Result_Data_64_bytes[60];
	PlcInputs.ST60_2_DM260_Result_Data_64_bytes[61] := HwInputs.ST60_2_DM260_Result_Data_64_bytes[61];
	PlcInputs.ST60_2_DM260_Result_Data_64_bytes[62] := HwInputs.ST60_2_DM260_Result_Data_64_bytes[62];
	PlcInputs.ST60_2_DM260_Result_Data_64_bytes[63] := HwInputs.ST60_2_DM260_Result_Data_64_bytes[63];
	PlcInputs.ST60_2_DM260_Result_Data_64_bytes[64] := HwInputs.ST60_2_DM260_Result_Data_64_bytes[64];
	PlcInputs.ST60_2_DM260_Result_Data_64_bytes[65] := HwInputs.ST60_2_DM260_Result_Data_64_bytes[65];
	PlcInputs.ST60_2_DM260_Result_Data_64_bytes[66] := HwInputs.ST60_2_DM260_Result_Data_64_bytes[66];
	PlcInputs.ST60_2_DM260_Result_Data_64_bytes[67] := HwInputs.ST60_2_DM260_Result_Data_64_bytes[67];
	PlcInputs.ST60_2_DM260_Result_Data_64_bytes[68] := HwInputs.ST60_2_DM260_Result_Data_64_bytes[68];
	PlcInputs.ST60_2_DM260_Result_Data_64_bytes[69] := HwInputs.ST60_2_DM260_Result_Data_64_bytes[69];
	PlcInputs.ST60_2_DM260_Result_Data_64_bytes[70] := HwInputs.ST60_2_DM260_Result_Data_64_bytes[70];
	PlcInputs.ST60_2_DM260_Result_Data_64_bytes[71] := HwInputs.ST60_2_DM260_Result_Data_64_bytes[71];
	PlcInputs.ST60_1_DM260_Acquisition_Status[0] := HwInputs.ST60_1_DM260_Acquisition_Status[0];
	PlcInputs.ST60_1_DM260_Acquisition_Status[1] := HwInputs.ST60_1_DM260_Acquisition_Status[1];
	PlcInputs.ST60_1_DM260_Acquisition_Status[2] := HwInputs.ST60_1_DM260_Acquisition_Status[2];
	PlcInputs.ST60_1_DM260_Results_Status := HwInputs.ST60_1_DM260_Results_Status;
	PlcInputs.ST60_1_DM260_Soft_Event_Control := HwInputs.ST60_1_DM260_Soft_Event_Control;
	PlcInputs.ST60_1_DM260_Result_Data_64_bytes[0] := HwInputs.ST60_1_DM260_Result_Data_64_bytes[0];
	PlcInputs.ST60_1_DM260_Result_Data_64_bytes[1] := HwInputs.ST60_1_DM260_Result_Data_64_bytes[1];
	PlcInputs.ST60_1_DM260_Result_Data_64_bytes[2] := HwInputs.ST60_1_DM260_Result_Data_64_bytes[2];
	PlcInputs.ST60_1_DM260_Result_Data_64_bytes[3] := HwInputs.ST60_1_DM260_Result_Data_64_bytes[3];
	PlcInputs.ST60_1_DM260_Result_Data_64_bytes[4] := HwInputs.ST60_1_DM260_Result_Data_64_bytes[4];
	PlcInputs.ST60_1_DM260_Result_Data_64_bytes[5] := HwInputs.ST60_1_DM260_Result_Data_64_bytes[5];
	PlcInputs.ST60_1_DM260_Result_Data_64_bytes[6] := HwInputs.ST60_1_DM260_Result_Data_64_bytes[6];
	PlcInputs.ST60_1_DM260_Result_Data_64_bytes[7] := HwInputs.ST60_1_DM260_Result_Data_64_bytes[7];
	PlcInputs.ST60_1_DM260_Result_Data_64_bytes[8] := HwInputs.ST60_1_DM260_Result_Data_64_bytes[8];
	PlcInputs.ST60_1_DM260_Result_Data_64_bytes[9] := HwInputs.ST60_1_DM260_Result_Data_64_bytes[9];
	PlcInputs.ST60_1_DM260_Result_Data_64_bytes[10] := HwInputs.ST60_1_DM260_Result_Data_64_bytes[10];
	PlcInputs.ST60_1_DM260_Result_Data_64_bytes[11] := HwInputs.ST60_1_DM260_Result_Data_64_bytes[11];
	PlcInputs.ST60_1_DM260_Result_Data_64_bytes[12] := HwInputs.ST60_1_DM260_Result_Data_64_bytes[12];
	PlcInputs.ST60_1_DM260_Result_Data_64_bytes[13] := HwInputs.ST60_1_DM260_Result_Data_64_bytes[13];
	PlcInputs.ST60_1_DM260_Result_Data_64_bytes[14] := HwInputs.ST60_1_DM260_Result_Data_64_bytes[14];
	PlcInputs.ST60_1_DM260_Result_Data_64_bytes[15] := HwInputs.ST60_1_DM260_Result_Data_64_bytes[15];
	PlcInputs.ST60_1_DM260_Result_Data_64_bytes[16] := HwInputs.ST60_1_DM260_Result_Data_64_bytes[16];
	PlcInputs.ST60_1_DM260_Result_Data_64_bytes[17] := HwInputs.ST60_1_DM260_Result_Data_64_bytes[17];
	PlcInputs.ST60_1_DM260_Result_Data_64_bytes[18] := HwInputs.ST60_1_DM260_Result_Data_64_bytes[18];
	PlcInputs.ST60_1_DM260_Result_Data_64_bytes[19] := HwInputs.ST60_1_DM260_Result_Data_64_bytes[19];
	PlcInputs.ST60_1_DM260_Result_Data_64_bytes[20] := HwInputs.ST60_1_DM260_Result_Data_64_bytes[20];
	PlcInputs.ST60_1_DM260_Result_Data_64_bytes[21] := HwInputs.ST60_1_DM260_Result_Data_64_bytes[21];
	PlcInputs.ST60_1_DM260_Result_Data_64_bytes[22] := HwInputs.ST60_1_DM260_Result_Data_64_bytes[22];
	PlcInputs.ST60_1_DM260_Result_Data_64_bytes[23] := HwInputs.ST60_1_DM260_Result_Data_64_bytes[23];
	PlcInputs.ST60_1_DM260_Result_Data_64_bytes[24] := HwInputs.ST60_1_DM260_Result_Data_64_bytes[24];
	PlcInputs.ST60_1_DM260_Result_Data_64_bytes[25] := HwInputs.ST60_1_DM260_Result_Data_64_bytes[25];
	PlcInputs.ST60_1_DM260_Result_Data_64_bytes[26] := HwInputs.ST60_1_DM260_Result_Data_64_bytes[26];
	PlcInputs.ST60_1_DM260_Result_Data_64_bytes[27] := HwInputs.ST60_1_DM260_Result_Data_64_bytes[27];
	PlcInputs.ST60_1_DM260_Result_Data_64_bytes[28] := HwInputs.ST60_1_DM260_Result_Data_64_bytes[28];
	PlcInputs.ST60_1_DM260_Result_Data_64_bytes[29] := HwInputs.ST60_1_DM260_Result_Data_64_bytes[29];
	PlcInputs.ST60_1_DM260_Result_Data_64_bytes[30] := HwInputs.ST60_1_DM260_Result_Data_64_bytes[30];
	PlcInputs.ST60_1_DM260_Result_Data_64_bytes[31] := HwInputs.ST60_1_DM260_Result_Data_64_bytes[31];
	PlcInputs.ST60_1_DM260_Result_Data_64_bytes[32] := HwInputs.ST60_1_DM260_Result_Data_64_bytes[32];
	PlcInputs.ST60_1_DM260_Result_Data_64_bytes[33] := HwInputs.ST60_1_DM260_Result_Data_64_bytes[33];
	PlcInputs.ST60_1_DM260_Result_Data_64_bytes[34] := HwInputs.ST60_1_DM260_Result_Data_64_bytes[34];
	PlcInputs.ST60_1_DM260_Result_Data_64_bytes[35] := HwInputs.ST60_1_DM260_Result_Data_64_bytes[35];
	PlcInputs.ST60_1_DM260_Result_Data_64_bytes[36] := HwInputs.ST60_1_DM260_Result_Data_64_bytes[36];
	PlcInputs.ST60_1_DM260_Result_Data_64_bytes[37] := HwInputs.ST60_1_DM260_Result_Data_64_bytes[37];
	PlcInputs.ST60_1_DM260_Result_Data_64_bytes[38] := HwInputs.ST60_1_DM260_Result_Data_64_bytes[38];
	PlcInputs.ST60_1_DM260_Result_Data_64_bytes[39] := HwInputs.ST60_1_DM260_Result_Data_64_bytes[39];
	PlcInputs.ST60_1_DM260_Result_Data_64_bytes[40] := HwInputs.ST60_1_DM260_Result_Data_64_bytes[40];
	PlcInputs.ST60_1_DM260_Result_Data_64_bytes[41] := HwInputs.ST60_1_DM260_Result_Data_64_bytes[41];
	PlcInputs.ST60_1_DM260_Result_Data_64_bytes[42] := HwInputs.ST60_1_DM260_Result_Data_64_bytes[42];
	PlcInputs.ST60_1_DM260_Result_Data_64_bytes[43] := HwInputs.ST60_1_DM260_Result_Data_64_bytes[43];
	PlcInputs.ST60_1_DM260_Result_Data_64_bytes[44] := HwInputs.ST60_1_DM260_Result_Data_64_bytes[44];
	PlcInputs.ST60_1_DM260_Result_Data_64_bytes[45] := HwInputs.ST60_1_DM260_Result_Data_64_bytes[45];
	PlcInputs.ST60_1_DM260_Result_Data_64_bytes[46] := HwInputs.ST60_1_DM260_Result_Data_64_bytes[46];
	PlcInputs.ST60_1_DM260_Result_Data_64_bytes[47] := HwInputs.ST60_1_DM260_Result_Data_64_bytes[47];
	PlcInputs.ST60_1_DM260_Result_Data_64_bytes[48] := HwInputs.ST60_1_DM260_Result_Data_64_bytes[48];
	PlcInputs.ST60_1_DM260_Result_Data_64_bytes[49] := HwInputs.ST60_1_DM260_Result_Data_64_bytes[49];
	PlcInputs.ST60_1_DM260_Result_Data_64_bytes[50] := HwInputs.ST60_1_DM260_Result_Data_64_bytes[50];
	PlcInputs.ST60_1_DM260_Result_Data_64_bytes[51] := HwInputs.ST60_1_DM260_Result_Data_64_bytes[51];
	PlcInputs.ST60_1_DM260_Result_Data_64_bytes[52] := HwInputs.ST60_1_DM260_Result_Data_64_bytes[52];
	PlcInputs.ST60_1_DM260_Result_Data_64_bytes[53] := HwInputs.ST60_1_DM260_Result_Data_64_bytes[53];
	PlcInputs.ST60_1_DM260_Result_Data_64_bytes[54] := HwInputs.ST60_1_DM260_Result_Data_64_bytes[54];
	PlcInputs.ST60_1_DM260_Result_Data_64_bytes[55] := HwInputs.ST60_1_DM260_Result_Data_64_bytes[55];
	PlcInputs.ST60_1_DM260_Result_Data_64_bytes[56] := HwInputs.ST60_1_DM260_Result_Data_64_bytes[56];
	PlcInputs.ST60_1_DM260_Result_Data_64_bytes[57] := HwInputs.ST60_1_DM260_Result_Data_64_bytes[57];
	PlcInputs.ST60_1_DM260_Result_Data_64_bytes[58] := HwInputs.ST60_1_DM260_Result_Data_64_bytes[58];
	PlcInputs.ST60_1_DM260_Result_Data_64_bytes[59] := HwInputs.ST60_1_DM260_Result_Data_64_bytes[59];
	PlcInputs.ST60_1_DM260_Result_Data_64_bytes[60] := HwInputs.ST60_1_DM260_Result_Data_64_bytes[60];
	PlcInputs.ST60_1_DM260_Result_Data_64_bytes[61] := HwInputs.ST60_1_DM260_Result_Data_64_bytes[61];
	PlcInputs.ST60_1_DM260_Result_Data_64_bytes[62] := HwInputs.ST60_1_DM260_Result_Data_64_bytes[62];
	PlcInputs.ST60_1_DM260_Result_Data_64_bytes[63] := HwInputs.ST60_1_DM260_Result_Data_64_bytes[63];
	PlcInputs.ST60_1_DM260_Result_Data_64_bytes[64] := HwInputs.ST60_1_DM260_Result_Data_64_bytes[64];
	PlcInputs.ST60_1_DM260_Result_Data_64_bytes[65] := HwInputs.ST60_1_DM260_Result_Data_64_bytes[65];
	PlcInputs.ST60_1_DM260_Result_Data_64_bytes[66] := HwInputs.ST60_1_DM260_Result_Data_64_bytes[66];
	PlcInputs.ST60_1_DM260_Result_Data_64_bytes[67] := HwInputs.ST60_1_DM260_Result_Data_64_bytes[67];
	PlcInputs.ST60_1_DM260_Result_Data_64_bytes[68] := HwInputs.ST60_1_DM260_Result_Data_64_bytes[68];
	PlcInputs.ST60_1_DM260_Result_Data_64_bytes[69] := HwInputs.ST60_1_DM260_Result_Data_64_bytes[69];
	PlcInputs.ST60_1_DM260_Result_Data_64_bytes[70] := HwInputs.ST60_1_DM260_Result_Data_64_bytes[70];
	PlcInputs.ST60_1_DM260_Result_Data_64_bytes[71] := HwInputs.ST60_1_DM260_Result_Data_64_bytes[71];
	PlcInputs.ST60_1_DM260_WPC_Acquisition_Status[0] := HwInputs.ST60_1_DM260_WPC_Acquisition_Status[0];
	PlcInputs.ST60_1_DM260_WPC_Acquisition_Status[1] := HwInputs.ST60_1_DM260_WPC_Acquisition_Status[1];
	PlcInputs.ST60_1_DM260_WPC_Acquisition_Status[2] := HwInputs.ST60_1_DM260_WPC_Acquisition_Status[2];
	PlcInputs.ST60_1_DM260_WPC_Results_Status := HwInputs.ST60_1_DM260_WPC_Results_Status;
	PlcInputs.ST60_1_DM260_WPC_Soft_Event_Control := HwInputs.ST60_1_DM260_WPC_Soft_Event_Control;
	PlcInputs.ST60_1_DM260_WPC_Result_Data_64_bytes[0] := HwInputs.ST60_1_DM260_WPC_Result_Data_64_bytes[0];
	PlcInputs.ST60_1_DM260_WPC_Result_Data_64_bytes[1] := HwInputs.ST60_1_DM260_WPC_Result_Data_64_bytes[1];
	PlcInputs.ST60_1_DM260_WPC_Result_Data_64_bytes[2] := HwInputs.ST60_1_DM260_WPC_Result_Data_64_bytes[2];
	PlcInputs.ST60_1_DM260_WPC_Result_Data_64_bytes[3] := HwInputs.ST60_1_DM260_WPC_Result_Data_64_bytes[3];
	PlcInputs.ST60_1_DM260_WPC_Result_Data_64_bytes[4] := HwInputs.ST60_1_DM260_WPC_Result_Data_64_bytes[4];
	PlcInputs.ST60_1_DM260_WPC_Result_Data_64_bytes[5] := HwInputs.ST60_1_DM260_WPC_Result_Data_64_bytes[5];
	PlcInputs.ST60_1_DM260_WPC_Result_Data_64_bytes[6] := HwInputs.ST60_1_DM260_WPC_Result_Data_64_bytes[6];
	PlcInputs.ST60_1_DM260_WPC_Result_Data_64_bytes[7] := HwInputs.ST60_1_DM260_WPC_Result_Data_64_bytes[7];
	PlcInputs.ST60_1_DM260_WPC_Result_Data_64_bytes[8] := HwInputs.ST60_1_DM260_WPC_Result_Data_64_bytes[8];
	PlcInputs.ST60_1_DM260_WPC_Result_Data_64_bytes[9] := HwInputs.ST60_1_DM260_WPC_Result_Data_64_bytes[9];
	PlcInputs.ST60_1_DM260_WPC_Result_Data_64_bytes[10] := HwInputs.ST60_1_DM260_WPC_Result_Data_64_bytes[10];
	PlcInputs.ST60_1_DM260_WPC_Result_Data_64_bytes[11] := HwInputs.ST60_1_DM260_WPC_Result_Data_64_bytes[11];
	PlcInputs.ST60_1_DM260_WPC_Result_Data_64_bytes[12] := HwInputs.ST60_1_DM260_WPC_Result_Data_64_bytes[12];
	PlcInputs.ST60_1_DM260_WPC_Result_Data_64_bytes[13] := HwInputs.ST60_1_DM260_WPC_Result_Data_64_bytes[13];
	PlcInputs.ST60_1_DM260_WPC_Result_Data_64_bytes[14] := HwInputs.ST60_1_DM260_WPC_Result_Data_64_bytes[14];
	PlcInputs.ST60_1_DM260_WPC_Result_Data_64_bytes[15] := HwInputs.ST60_1_DM260_WPC_Result_Data_64_bytes[15];
	PlcInputs.ST60_1_DM260_WPC_Result_Data_64_bytes[16] := HwInputs.ST60_1_DM260_WPC_Result_Data_64_bytes[16];
	PlcInputs.ST60_1_DM260_WPC_Result_Data_64_bytes[17] := HwInputs.ST60_1_DM260_WPC_Result_Data_64_bytes[17];
	PlcInputs.ST60_1_DM260_WPC_Result_Data_64_bytes[18] := HwInputs.ST60_1_DM260_WPC_Result_Data_64_bytes[18];
	PlcInputs.ST60_1_DM260_WPC_Result_Data_64_bytes[19] := HwInputs.ST60_1_DM260_WPC_Result_Data_64_bytes[19];
	PlcInputs.ST60_1_DM260_WPC_Result_Data_64_bytes[20] := HwInputs.ST60_1_DM260_WPC_Result_Data_64_bytes[20];
	PlcInputs.ST60_1_DM260_WPC_Result_Data_64_bytes[21] := HwInputs.ST60_1_DM260_WPC_Result_Data_64_bytes[21];
	PlcInputs.ST60_1_DM260_WPC_Result_Data_64_bytes[22] := HwInputs.ST60_1_DM260_WPC_Result_Data_64_bytes[22];
	PlcInputs.ST60_1_DM260_WPC_Result_Data_64_bytes[23] := HwInputs.ST60_1_DM260_WPC_Result_Data_64_bytes[23];
	PlcInputs.ST60_1_DM260_WPC_Result_Data_64_bytes[24] := HwInputs.ST60_1_DM260_WPC_Result_Data_64_bytes[24];
	PlcInputs.ST60_1_DM260_WPC_Result_Data_64_bytes[25] := HwInputs.ST60_1_DM260_WPC_Result_Data_64_bytes[25];
	PlcInputs.ST60_1_DM260_WPC_Result_Data_64_bytes[26] := HwInputs.ST60_1_DM260_WPC_Result_Data_64_bytes[26];
	PlcInputs.ST60_1_DM260_WPC_Result_Data_64_bytes[27] := HwInputs.ST60_1_DM260_WPC_Result_Data_64_bytes[27];
	PlcInputs.ST60_1_DM260_WPC_Result_Data_64_bytes[28] := HwInputs.ST60_1_DM260_WPC_Result_Data_64_bytes[28];
	PlcInputs.ST60_1_DM260_WPC_Result_Data_64_bytes[29] := HwInputs.ST60_1_DM260_WPC_Result_Data_64_bytes[29];
	PlcInputs.ST60_1_DM260_WPC_Result_Data_64_bytes[30] := HwInputs.ST60_1_DM260_WPC_Result_Data_64_bytes[30];
	PlcInputs.ST60_1_DM260_WPC_Result_Data_64_bytes[31] := HwInputs.ST60_1_DM260_WPC_Result_Data_64_bytes[31];
	PlcInputs.ST60_1_DM260_WPC_Result_Data_64_bytes[32] := HwInputs.ST60_1_DM260_WPC_Result_Data_64_bytes[32];
	PlcInputs.ST60_1_DM260_WPC_Result_Data_64_bytes[33] := HwInputs.ST60_1_DM260_WPC_Result_Data_64_bytes[33];
	PlcInputs.ST60_1_DM260_WPC_Result_Data_64_bytes[34] := HwInputs.ST60_1_DM260_WPC_Result_Data_64_bytes[34];
	PlcInputs.ST60_1_DM260_WPC_Result_Data_64_bytes[35] := HwInputs.ST60_1_DM260_WPC_Result_Data_64_bytes[35];
	PlcInputs.ST60_1_DM260_WPC_Result_Data_64_bytes[36] := HwInputs.ST60_1_DM260_WPC_Result_Data_64_bytes[36];
	PlcInputs.ST60_1_DM260_WPC_Result_Data_64_bytes[37] := HwInputs.ST60_1_DM260_WPC_Result_Data_64_bytes[37];
	PlcInputs.ST60_1_DM260_WPC_Result_Data_64_bytes[38] := HwInputs.ST60_1_DM260_WPC_Result_Data_64_bytes[38];
	PlcInputs.ST60_1_DM260_WPC_Result_Data_64_bytes[39] := HwInputs.ST60_1_DM260_WPC_Result_Data_64_bytes[39];
	PlcInputs.ST60_1_DM260_WPC_Result_Data_64_bytes[40] := HwInputs.ST60_1_DM260_WPC_Result_Data_64_bytes[40];
	PlcInputs.ST60_1_DM260_WPC_Result_Data_64_bytes[41] := HwInputs.ST60_1_DM260_WPC_Result_Data_64_bytes[41];
	PlcInputs.ST60_1_DM260_WPC_Result_Data_64_bytes[42] := HwInputs.ST60_1_DM260_WPC_Result_Data_64_bytes[42];
	PlcInputs.ST60_1_DM260_WPC_Result_Data_64_bytes[43] := HwInputs.ST60_1_DM260_WPC_Result_Data_64_bytes[43];
	PlcInputs.ST60_1_DM260_WPC_Result_Data_64_bytes[44] := HwInputs.ST60_1_DM260_WPC_Result_Data_64_bytes[44];
	PlcInputs.ST60_1_DM260_WPC_Result_Data_64_bytes[45] := HwInputs.ST60_1_DM260_WPC_Result_Data_64_bytes[45];
	PlcInputs.ST60_1_DM260_WPC_Result_Data_64_bytes[46] := HwInputs.ST60_1_DM260_WPC_Result_Data_64_bytes[46];
	PlcInputs.ST60_1_DM260_WPC_Result_Data_64_bytes[47] := HwInputs.ST60_1_DM260_WPC_Result_Data_64_bytes[47];
	PlcInputs.ST60_1_DM260_WPC_Result_Data_64_bytes[48] := HwInputs.ST60_1_DM260_WPC_Result_Data_64_bytes[48];
	PlcInputs.ST60_1_DM260_WPC_Result_Data_64_bytes[49] := HwInputs.ST60_1_DM260_WPC_Result_Data_64_bytes[49];
	PlcInputs.ST60_1_DM260_WPC_Result_Data_64_bytes[50] := HwInputs.ST60_1_DM260_WPC_Result_Data_64_bytes[50];
	PlcInputs.ST60_1_DM260_WPC_Result_Data_64_bytes[51] := HwInputs.ST60_1_DM260_WPC_Result_Data_64_bytes[51];
	PlcInputs.ST60_1_DM260_WPC_Result_Data_64_bytes[52] := HwInputs.ST60_1_DM260_WPC_Result_Data_64_bytes[52];
	PlcInputs.ST60_1_DM260_WPC_Result_Data_64_bytes[53] := HwInputs.ST60_1_DM260_WPC_Result_Data_64_bytes[53];
	PlcInputs.ST60_1_DM260_WPC_Result_Data_64_bytes[54] := HwInputs.ST60_1_DM260_WPC_Result_Data_64_bytes[54];
	PlcInputs.ST60_1_DM260_WPC_Result_Data_64_bytes[55] := HwInputs.ST60_1_DM260_WPC_Result_Data_64_bytes[55];
	PlcInputs.ST60_1_DM260_WPC_Result_Data_64_bytes[56] := HwInputs.ST60_1_DM260_WPC_Result_Data_64_bytes[56];
	PlcInputs.ST60_1_DM260_WPC_Result_Data_64_bytes[57] := HwInputs.ST60_1_DM260_WPC_Result_Data_64_bytes[57];
	PlcInputs.ST60_1_DM260_WPC_Result_Data_64_bytes[58] := HwInputs.ST60_1_DM260_WPC_Result_Data_64_bytes[58];
	PlcInputs.ST60_1_DM260_WPC_Result_Data_64_bytes[59] := HwInputs.ST60_1_DM260_WPC_Result_Data_64_bytes[59];
	PlcInputs.ST60_1_DM260_WPC_Result_Data_64_bytes[60] := HwInputs.ST60_1_DM260_WPC_Result_Data_64_bytes[60];
	PlcInputs.ST60_1_DM260_WPC_Result_Data_64_bytes[61] := HwInputs.ST60_1_DM260_WPC_Result_Data_64_bytes[61];
	PlcInputs.ST60_1_DM260_WPC_Result_Data_64_bytes[62] := HwInputs.ST60_1_DM260_WPC_Result_Data_64_bytes[62];
	PlcInputs.ST60_1_DM260_WPC_Result_Data_64_bytes[63] := HwInputs.ST60_1_DM260_WPC_Result_Data_64_bytes[63];
	PlcInputs.ST60_1_DM260_WPC_Result_Data_64_bytes[64] := HwInputs.ST60_1_DM260_WPC_Result_Data_64_bytes[64];
	PlcInputs.ST60_1_DM260_WPC_Result_Data_64_bytes[65] := HwInputs.ST60_1_DM260_WPC_Result_Data_64_bytes[65];
	PlcInputs.ST60_1_DM260_WPC_Result_Data_64_bytes[66] := HwInputs.ST60_1_DM260_WPC_Result_Data_64_bytes[66];
	PlcInputs.ST60_1_DM260_WPC_Result_Data_64_bytes[67] := HwInputs.ST60_1_DM260_WPC_Result_Data_64_bytes[67];
	PlcInputs.ST60_1_DM260_WPC_Result_Data_64_bytes[68] := HwInputs.ST60_1_DM260_WPC_Result_Data_64_bytes[68];
	PlcInputs.ST60_1_DM260_WPC_Result_Data_64_bytes[69] := HwInputs.ST60_1_DM260_WPC_Result_Data_64_bytes[69];
	PlcInputs.ST60_1_DM260_WPC_Result_Data_64_bytes[70] := HwInputs.ST60_1_DM260_WPC_Result_Data_64_bytes[70];
	PlcInputs.ST60_1_DM260_WPC_Result_Data_64_bytes[71] := HwInputs.ST60_1_DM260_WPC_Result_Data_64_bytes[71];
	PlcInputs.ST60_TZ535_PN_In_Out_32_byte_x[0] := HwInputs.ST60_TZ535_PN_In_Out_32_byte_x[0];
	PlcInputs.ST60_TZ535_PN_In_Out_32_byte_x[1] := HwInputs.ST60_TZ535_PN_In_Out_32_byte_x[1];
	PlcInputs.ST60_TZ535_PN_In_Out_32_byte_x[2] := HwInputs.ST60_TZ535_PN_In_Out_32_byte_x[2];
	PlcInputs.ST60_TZ535_PN_In_Out_32_byte_x[3] := HwInputs.ST60_TZ535_PN_In_Out_32_byte_x[3];
	PlcInputs.ST60_TZ535_PN_In_Out_32_byte_x[4] := HwInputs.ST60_TZ535_PN_In_Out_32_byte_x[4];
	PlcInputs.ST60_TZ535_PN_In_Out_32_byte_x[5] := HwInputs.ST60_TZ535_PN_In_Out_32_byte_x[5];
	PlcInputs.ST60_TZ535_PN_In_Out_32_byte_x[6] := HwInputs.ST60_TZ535_PN_In_Out_32_byte_x[6];
	PlcInputs.ST60_TZ535_PN_In_Out_32_byte_x[7] := HwInputs.ST60_TZ535_PN_In_Out_32_byte_x[7];
	PlcInputs.ST60_TZ535_PN_In_Out_32_byte_x[8] := HwInputs.ST60_TZ535_PN_In_Out_32_byte_x[8];
	PlcInputs.ST60_TZ535_PN_In_Out_32_byte_x[9] := HwInputs.ST60_TZ535_PN_In_Out_32_byte_x[9];
	PlcInputs.ST60_TZ535_PN_In_Out_32_byte_x[10] := HwInputs.ST60_TZ535_PN_In_Out_32_byte_x[10];
	PlcInputs.ST60_TZ535_PN_In_Out_32_byte_x[11] := HwInputs.ST60_TZ535_PN_In_Out_32_byte_x[11];
	PlcInputs.ST60_TZ535_PN_In_Out_32_byte_x[12] := HwInputs.ST60_TZ535_PN_In_Out_32_byte_x[12];
	PlcInputs.ST60_TZ535_PN_In_Out_32_byte_x[13] := HwInputs.ST60_TZ535_PN_In_Out_32_byte_x[13];
	PlcInputs.ST60_TZ535_PN_In_Out_32_byte_x[14] := HwInputs.ST60_TZ535_PN_In_Out_32_byte_x[14];
	PlcInputs.ST60_TZ535_PN_In_Out_32_byte_x[15] := HwInputs.ST60_TZ535_PN_In_Out_32_byte_x[15];
	PlcInputs.ST60_TZ535_PN_In_Out_32_byte_x[16] := HwInputs.ST60_TZ535_PN_In_Out_32_byte_x[16];
	PlcInputs.ST60_TZ535_PN_In_Out_32_byte_x[17] := HwInputs.ST60_TZ535_PN_In_Out_32_byte_x[17];
	PlcInputs.ST60_TZ535_PN_In_Out_32_byte_x[18] := HwInputs.ST60_TZ535_PN_In_Out_32_byte_x[18];
	PlcInputs.ST60_TZ535_PN_In_Out_32_byte_x[19] := HwInputs.ST60_TZ535_PN_In_Out_32_byte_x[19];
	PlcInputs.ST60_TZ535_PN_In_Out_32_byte_x[20] := HwInputs.ST60_TZ535_PN_In_Out_32_byte_x[20];
	PlcInputs.ST60_TZ535_PN_In_Out_32_byte_x[21] := HwInputs.ST60_TZ535_PN_In_Out_32_byte_x[21];
	PlcInputs.ST60_TZ535_PN_In_Out_32_byte_x[22] := HwInputs.ST60_TZ535_PN_In_Out_32_byte_x[22];
	PlcInputs.ST60_TZ535_PN_In_Out_32_byte_x[23] := HwInputs.ST60_TZ535_PN_In_Out_32_byte_x[23];
	PlcInputs.ST60_TZ535_PN_In_Out_32_byte_x[24] := HwInputs.ST60_TZ535_PN_In_Out_32_byte_x[24];
	PlcInputs.ST60_TZ535_PN_In_Out_32_byte_x[25] := HwInputs.ST60_TZ535_PN_In_Out_32_byte_x[25];
	PlcInputs.ST60_TZ535_PN_In_Out_32_byte_x[26] := HwInputs.ST60_TZ535_PN_In_Out_32_byte_x[26];
	PlcInputs.ST60_TZ535_PN_In_Out_32_byte_x[27] := HwInputs.ST60_TZ535_PN_In_Out_32_byte_x[27];
	PlcInputs.ST60_TZ535_PN_In_Out_32_byte_x[28] := HwInputs.ST60_TZ535_PN_In_Out_32_byte_x[28];
	PlcInputs.ST60_TZ535_PN_In_Out_32_byte_x[29] := HwInputs.ST60_TZ535_PN_In_Out_32_byte_x[29];
	PlcInputs.ST60_TZ535_PN_In_Out_32_byte_x[30] := HwInputs.ST60_TZ535_PN_In_Out_32_byte_x[30];
	PlcInputs.ST60_TZ535_PN_In_Out_32_byte_x[31] := HwInputs.ST60_TZ535_PN_In_Out_32_byte_x[31];
	PlcInputs.ST60_SCHUNK_R_IN_4_Double_Words[0] := HwInputs.ST60_SCHUNK_R_IN_4_Double_Words[0];
	PlcInputs.ST60_SCHUNK_R_IN_4_Double_Words[1] := HwInputs.ST60_SCHUNK_R_IN_4_Double_Words[1];
	PlcInputs.ST60_SCHUNK_R_IN_4_Double_Words[2] := HwInputs.ST60_SCHUNK_R_IN_4_Double_Words[2];
	PlcInputs.ST60_SCHUNK_R_IN_4_Double_Words[3] := HwInputs.ST60_SCHUNK_R_IN_4_Double_Words[3];
	PlcInputs.ST60_SCHUNK_R_IN_4_Double_Words[4] := HwInputs.ST60_SCHUNK_R_IN_4_Double_Words[4];
	PlcInputs.ST60_SCHUNK_R_IN_4_Double_Words[5] := HwInputs.ST60_SCHUNK_R_IN_4_Double_Words[5];
	PlcInputs.ST60_SCHUNK_R_IN_4_Double_Words[6] := HwInputs.ST60_SCHUNK_R_IN_4_Double_Words[6];
	PlcInputs.ST60_SCHUNK_R_IN_4_Double_Words[7] := HwInputs.ST60_SCHUNK_R_IN_4_Double_Words[7];
	PlcInputs.ST60_SCHUNK_R_IN_4_Double_Words[8] := HwInputs.ST60_SCHUNK_R_IN_4_Double_Words[8];
	PlcInputs.ST60_SCHUNK_R_IN_4_Double_Words[9] := HwInputs.ST60_SCHUNK_R_IN_4_Double_Words[9];
	PlcInputs.ST60_SCHUNK_R_IN_4_Double_Words[10] := HwInputs.ST60_SCHUNK_R_IN_4_Double_Words[10];
	PlcInputs.ST60_SCHUNK_R_IN_4_Double_Words[11] := HwInputs.ST60_SCHUNK_R_IN_4_Double_Words[11];
	PlcInputs.ST60_SCHUNK_R_IN_4_Double_Words[12] := HwInputs.ST60_SCHUNK_R_IN_4_Double_Words[12];
	PlcInputs.ST60_SCHUNK_R_IN_4_Double_Words[13] := HwInputs.ST60_SCHUNK_R_IN_4_Double_Words[13];
	PlcInputs.ST60_SCHUNK_R_IN_4_Double_Words[14] := HwInputs.ST60_SCHUNK_R_IN_4_Double_Words[14];
	PlcInputs.ST60_SCHUNK_R_IN_4_Double_Words[15] := HwInputs.ST60_SCHUNK_R_IN_4_Double_Words[15];
	PlcInputs.ST60_SCHUNK_L_IN_4_Double_Words[0] := HwInputs.ST60_SCHUNK_L_IN_4_Double_Words[0];
	PlcInputs.ST60_SCHUNK_L_IN_4_Double_Words[1] := HwInputs.ST60_SCHUNK_L_IN_4_Double_Words[1];
	PlcInputs.ST60_SCHUNK_L_IN_4_Double_Words[2] := HwInputs.ST60_SCHUNK_L_IN_4_Double_Words[2];
	PlcInputs.ST60_SCHUNK_L_IN_4_Double_Words[3] := HwInputs.ST60_SCHUNK_L_IN_4_Double_Words[3];
	PlcInputs.ST60_SCHUNK_L_IN_4_Double_Words[4] := HwInputs.ST60_SCHUNK_L_IN_4_Double_Words[4];
	PlcInputs.ST60_SCHUNK_L_IN_4_Double_Words[5] := HwInputs.ST60_SCHUNK_L_IN_4_Double_Words[5];
	PlcInputs.ST60_SCHUNK_L_IN_4_Double_Words[6] := HwInputs.ST60_SCHUNK_L_IN_4_Double_Words[6];
	PlcInputs.ST60_SCHUNK_L_IN_4_Double_Words[7] := HwInputs.ST60_SCHUNK_L_IN_4_Double_Words[7];
	PlcInputs.ST60_SCHUNK_L_IN_4_Double_Words[8] := HwInputs.ST60_SCHUNK_L_IN_4_Double_Words[8];
	PlcInputs.ST60_SCHUNK_L_IN_4_Double_Words[9] := HwInputs.ST60_SCHUNK_L_IN_4_Double_Words[9];
	PlcInputs.ST60_SCHUNK_L_IN_4_Double_Words[10] := HwInputs.ST60_SCHUNK_L_IN_4_Double_Words[10];
	PlcInputs.ST60_SCHUNK_L_IN_4_Double_Words[11] := HwInputs.ST60_SCHUNK_L_IN_4_Double_Words[11];
	PlcInputs.ST60_SCHUNK_L_IN_4_Double_Words[12] := HwInputs.ST60_SCHUNK_L_IN_4_Double_Words[12];
	PlcInputs.ST60_SCHUNK_L_IN_4_Double_Words[13] := HwInputs.ST60_SCHUNK_L_IN_4_Double_Words[13];
	PlcInputs.ST60_SCHUNK_L_IN_4_Double_Words[14] := HwInputs.ST60_SCHUNK_L_IN_4_Double_Words[14];
	PlcInputs.ST60_SCHUNK_L_IN_4_Double_Words[15] := HwInputs.ST60_SCHUNK_L_IN_4_Double_Words[15];
	PlcInputs.ST60_ET200SP_CM_4xIO_Link_1[0] := HwInputs.ST60_ET200SP_CM_4xIO_Link_1[0];
	PlcInputs.ST60_ET200SP_CM_4xIO_Link_1[1] := HwInputs.ST60_ET200SP_CM_4xIO_Link_1[1];
	PlcInputs.ST60_ET200SP_CM_4xIO_Link_1[2] := HwInputs.ST60_ET200SP_CM_4xIO_Link_1[2];
	PlcInputs.ST60_ET200SP_CM_4xIO_Link_1[3] := HwInputs.ST60_ET200SP_CM_4xIO_Link_1[3];
	PlcInputs.ST60_ET200SP_CM_4xIO_Link_1[4] := HwInputs.ST60_ET200SP_CM_4xIO_Link_1[4];
	PlcInputs.ST60_ET200SP_CM_4xIO_Link_1[5] := HwInputs.ST60_ET200SP_CM_4xIO_Link_1[5];
	PlcInputs.ST60_ET200SP_CM_4xIO_Link_1[6] := HwInputs.ST60_ET200SP_CM_4xIO_Link_1[6];
	PlcInputs.ST60_ET200SP_CM_4xIO_Link_1[7] := HwInputs.ST60_ET200SP_CM_4xIO_Link_1[7];
	PlcInputs.ST60_ET200SP_CM_4xIO_Link_1[8] := HwInputs.ST60_ET200SP_CM_4xIO_Link_1[8];
	PlcInputs.ST60_ET200SP_CM_4xIO_Link_1[9] := HwInputs.ST60_ET200SP_CM_4xIO_Link_1[9];
	PlcInputs.ST60_ET200SP_CM_4xIO_Link_1[10] := HwInputs.ST60_ET200SP_CM_4xIO_Link_1[10];
	PlcInputs.ST60_ET200SP_CM_4xIO_Link_1[11] := HwInputs.ST60_ET200SP_CM_4xIO_Link_1[11];
	PlcInputs.ST60_ET200SP_CM_4xIO_Link_1[12] := HwInputs.ST60_ET200SP_CM_4xIO_Link_1[12];
	PlcInputs.ST60_ET200SP_CM_4xIO_Link_1[13] := HwInputs.ST60_ET200SP_CM_4xIO_Link_1[13];
	PlcInputs.ST60_ET200SP_CM_4xIO_Link_1[14] := HwInputs.ST60_ET200SP_CM_4xIO_Link_1[14];
	PlcInputs.ST60_ET200SP_CM_4xIO_Link_1[15] := HwInputs.ST60_ET200SP_CM_4xIO_Link_1[15];
	PlcInputs.ST60_ET200SP_CM_4xIO_Link_1[16] := HwInputs.ST60_ET200SP_CM_4xIO_Link_1[16];
	PlcInputs.ST60_ET200SP_CM_4xIO_Link_1[17] := HwInputs.ST60_ET200SP_CM_4xIO_Link_1[17];
	PlcInputs.ST60_ET200SP_CM_4xIO_Link_1[18] := HwInputs.ST60_ET200SP_CM_4xIO_Link_1[18];
	PlcInputs.ST60_ET200SP_CM_4xIO_Link_1[19] := HwInputs.ST60_ET200SP_CM_4xIO_Link_1[19];
	PlcInputs.ST60_ET200SP_CM_4xIO_Link_1[20] := HwInputs.ST60_ET200SP_CM_4xIO_Link_1[20];
	PlcInputs.ST60_ET200SP_CM_4xIO_Link_1[21] := HwInputs.ST60_ET200SP_CM_4xIO_Link_1[21];
	PlcInputs.ST60_ET200SP_CM_4xIO_Link_1[22] := HwInputs.ST60_ET200SP_CM_4xIO_Link_1[22];
	PlcInputs.ST60_ET200SP_CM_4xIO_Link_1[23] := HwInputs.ST60_ET200SP_CM_4xIO_Link_1[23];
	PlcInputs.ST60_ET200SP_CM_4xIO_Link_1[24] := HwInputs.ST60_ET200SP_CM_4xIO_Link_1[24];
	PlcInputs.ST60_ET200SP_CM_4xIO_Link_1[25] := HwInputs.ST60_ET200SP_CM_4xIO_Link_1[25];
	PlcInputs.ST60_ET200SP_CM_4xIO_Link_1[26] := HwInputs.ST60_ET200SP_CM_4xIO_Link_1[26];
	PlcInputs.ST60_ET200SP_CM_4xIO_Link_1[27] := HwInputs.ST60_ET200SP_CM_4xIO_Link_1[27];
	PlcInputs.ST60_ET200SP_CM_4xIO_Link_1[28] := HwInputs.ST60_ET200SP_CM_4xIO_Link_1[28];
	PlcInputs.ST60_ET200SP_CM_4xIO_Link_1[29] := HwInputs.ST60_ET200SP_CM_4xIO_Link_1[29];
	PlcInputs.ST60_ET200SP_CM_4xIO_Link_1[30] := HwInputs.ST60_ET200SP_CM_4xIO_Link_1[30];
	PlcInputs.ST60_ET200SP_CM_4xIO_Link_1[31] := HwInputs.ST60_ET200SP_CM_4xIO_Link_1[31];
	PlcInputs.ST60_ET200SP_CM_4xIO_Link_2[0] := HwInputs.ST60_ET200SP_CM_4xIO_Link_2[0];
	PlcInputs.ST60_ET200SP_CM_4xIO_Link_2[1] := HwInputs.ST60_ET200SP_CM_4xIO_Link_2[1];
	PlcInputs.ST60_ET200SP_CM_4xIO_Link_2[2] := HwInputs.ST60_ET200SP_CM_4xIO_Link_2[2];
	PlcInputs.ST60_ET200SP_CM_4xIO_Link_2[3] := HwInputs.ST60_ET200SP_CM_4xIO_Link_2[3];
	PlcInputs.ST60_ET200SP_CM_4xIO_Link_2[4] := HwInputs.ST60_ET200SP_CM_4xIO_Link_2[4];
	PlcInputs.ST60_ET200SP_CM_4xIO_Link_2[5] := HwInputs.ST60_ET200SP_CM_4xIO_Link_2[5];
	PlcInputs.ST60_ET200SP_CM_4xIO_Link_2[6] := HwInputs.ST60_ET200SP_CM_4xIO_Link_2[6];
	PlcInputs.ST60_ET200SP_CM_4xIO_Link_2[7] := HwInputs.ST60_ET200SP_CM_4xIO_Link_2[7];
	PlcInputs.ST60_ET200SP_CM_4xIO_Link_2[8] := HwInputs.ST60_ET200SP_CM_4xIO_Link_2[8];
	PlcInputs.ST60_ET200SP_CM_4xIO_Link_2[9] := HwInputs.ST60_ET200SP_CM_4xIO_Link_2[9];
	PlcInputs.ST60_ET200SP_CM_4xIO_Link_2[10] := HwInputs.ST60_ET200SP_CM_4xIO_Link_2[10];
	PlcInputs.ST60_ET200SP_CM_4xIO_Link_2[11] := HwInputs.ST60_ET200SP_CM_4xIO_Link_2[11];
	PlcInputs.ST60_ET200SP_CM_4xIO_Link_2[12] := HwInputs.ST60_ET200SP_CM_4xIO_Link_2[12];
	PlcInputs.ST60_ET200SP_CM_4xIO_Link_2[13] := HwInputs.ST60_ET200SP_CM_4xIO_Link_2[13];
	PlcInputs.ST60_ET200SP_CM_4xIO_Link_2[14] := HwInputs.ST60_ET200SP_CM_4xIO_Link_2[14];
	PlcInputs.ST60_ET200SP_CM_4xIO_Link_2[15] := HwInputs.ST60_ET200SP_CM_4xIO_Link_2[15];
	PlcInputs.ST60_ET200SP_CM_4xIO_Link_2[16] := HwInputs.ST60_ET200SP_CM_4xIO_Link_2[16];
	PlcInputs.ST60_ET200SP_CM_4xIO_Link_2[17] := HwInputs.ST60_ET200SP_CM_4xIO_Link_2[17];
	PlcInputs.ST60_ET200SP_CM_4xIO_Link_2[18] := HwInputs.ST60_ET200SP_CM_4xIO_Link_2[18];
	PlcInputs.ST60_ET200SP_CM_4xIO_Link_2[19] := HwInputs.ST60_ET200SP_CM_4xIO_Link_2[19];
	PlcInputs.ST60_ET200SP_CM_4xIO_Link_2[20] := HwInputs.ST60_ET200SP_CM_4xIO_Link_2[20];
	PlcInputs.ST60_ET200SP_CM_4xIO_Link_2[21] := HwInputs.ST60_ET200SP_CM_4xIO_Link_2[21];
	PlcInputs.ST60_ET200SP_CM_4xIO_Link_2[22] := HwInputs.ST60_ET200SP_CM_4xIO_Link_2[22];
	PlcInputs.ST60_ET200SP_CM_4xIO_Link_2[23] := HwInputs.ST60_ET200SP_CM_4xIO_Link_2[23];
	PlcInputs.ST60_ET200SP_CM_4xIO_Link_2[24] := HwInputs.ST60_ET200SP_CM_4xIO_Link_2[24];
	PlcInputs.ST60_ET200SP_CM_4xIO_Link_2[25] := HwInputs.ST60_ET200SP_CM_4xIO_Link_2[25];
	PlcInputs.ST60_ET200SP_CM_4xIO_Link_2[26] := HwInputs.ST60_ET200SP_CM_4xIO_Link_2[26];
	PlcInputs.ST60_ET200SP_CM_4xIO_Link_2[27] := HwInputs.ST60_ET200SP_CM_4xIO_Link_2[27];
	PlcInputs.ST60_ET200SP_CM_4xIO_Link_2[28] := HwInputs.ST60_ET200SP_CM_4xIO_Link_2[28];
	PlcInputs.ST60_ET200SP_CM_4xIO_Link_2[29] := HwInputs.ST60_ET200SP_CM_4xIO_Link_2[29];
	PlcInputs.ST60_ET200SP_CM_4xIO_Link_2[30] := HwInputs.ST60_ET200SP_CM_4xIO_Link_2[30];
	PlcInputs.ST60_ET200SP_CM_4xIO_Link_2[31] := HwInputs.ST60_ET200SP_CM_4xIO_Link_2[31];
	PlcInputs.ST60_ET200SP_CM_4xIO_Link_3[0] := HwInputs.ST60_ET200SP_CM_4xIO_Link_3[0];
	PlcInputs.ST60_ET200SP_CM_4xIO_Link_3[1] := HwInputs.ST60_ET200SP_CM_4xIO_Link_3[1];
	PlcInputs.ST60_ET200SP_CM_4xIO_Link_3[2] := HwInputs.ST60_ET200SP_CM_4xIO_Link_3[2];
	PlcInputs.ST60_ET200SP_CM_4xIO_Link_3[3] := HwInputs.ST60_ET200SP_CM_4xIO_Link_3[3];
	PlcInputs.ST60_ET200SP_CM_4xIO_Link_3[4] := HwInputs.ST60_ET200SP_CM_4xIO_Link_3[4];
	PlcInputs.ST60_ET200SP_CM_4xIO_Link_3[5] := HwInputs.ST60_ET200SP_CM_4xIO_Link_3[5];
	PlcInputs.ST60_ET200SP_CM_4xIO_Link_3[6] := HwInputs.ST60_ET200SP_CM_4xIO_Link_3[6];
	PlcInputs.ST60_ET200SP_CM_4xIO_Link_3[7] := HwInputs.ST60_ET200SP_CM_4xIO_Link_3[7];
	PlcInputs.ST60_ET200SP_CM_4xIO_Link_3[8] := HwInputs.ST60_ET200SP_CM_4xIO_Link_3[8];
	PlcInputs.ST60_ET200SP_CM_4xIO_Link_3[9] := HwInputs.ST60_ET200SP_CM_4xIO_Link_3[9];
	PlcInputs.ST60_ET200SP_CM_4xIO_Link_3[10] := HwInputs.ST60_ET200SP_CM_4xIO_Link_3[10];
	PlcInputs.ST60_ET200SP_CM_4xIO_Link_3[11] := HwInputs.ST60_ET200SP_CM_4xIO_Link_3[11];
	PlcInputs.ST60_ET200SP_CM_4xIO_Link_3[12] := HwInputs.ST60_ET200SP_CM_4xIO_Link_3[12];
	PlcInputs.ST60_ET200SP_CM_4xIO_Link_3[13] := HwInputs.ST60_ET200SP_CM_4xIO_Link_3[13];
	PlcInputs.ST60_ET200SP_CM_4xIO_Link_3[14] := HwInputs.ST60_ET200SP_CM_4xIO_Link_3[14];
	PlcInputs.ST60_ET200SP_CM_4xIO_Link_3[15] := HwInputs.ST60_ET200SP_CM_4xIO_Link_3[15];
	PlcInputs.ST60_ET200SP_CM_4xIO_Link_3[16] := HwInputs.ST60_ET200SP_CM_4xIO_Link_3[16];
	PlcInputs.ST60_ET200SP_CM_4xIO_Link_3[17] := HwInputs.ST60_ET200SP_CM_4xIO_Link_3[17];
	PlcInputs.ST60_ET200SP_CM_4xIO_Link_3[18] := HwInputs.ST60_ET200SP_CM_4xIO_Link_3[18];
	PlcInputs.ST60_ET200SP_CM_4xIO_Link_3[19] := HwInputs.ST60_ET200SP_CM_4xIO_Link_3[19];
	PlcInputs.ST60_ET200SP_CM_4xIO_Link_3[20] := HwInputs.ST60_ET200SP_CM_4xIO_Link_3[20];
	PlcInputs.ST60_ET200SP_CM_4xIO_Link_3[21] := HwInputs.ST60_ET200SP_CM_4xIO_Link_3[21];
	PlcInputs.ST60_ET200SP_CM_4xIO_Link_3[22] := HwInputs.ST60_ET200SP_CM_4xIO_Link_3[22];
	PlcInputs.ST60_ET200SP_CM_4xIO_Link_3[23] := HwInputs.ST60_ET200SP_CM_4xIO_Link_3[23];
	PlcInputs.ST60_ET200SP_CM_4xIO_Link_3[24] := HwInputs.ST60_ET200SP_CM_4xIO_Link_3[24];
	PlcInputs.ST60_ET200SP_CM_4xIO_Link_3[25] := HwInputs.ST60_ET200SP_CM_4xIO_Link_3[25];
	PlcInputs.ST60_ET200SP_CM_4xIO_Link_3[26] := HwInputs.ST60_ET200SP_CM_4xIO_Link_3[26];
	PlcInputs.ST60_ET200SP_CM_4xIO_Link_3[27] := HwInputs.ST60_ET200SP_CM_4xIO_Link_3[27];
	PlcInputs.ST60_ET200SP_CM_4xIO_Link_3[28] := HwInputs.ST60_ET200SP_CM_4xIO_Link_3[28];
	PlcInputs.ST60_ET200SP_CM_4xIO_Link_3[29] := HwInputs.ST60_ET200SP_CM_4xIO_Link_3[29];
	PlcInputs.ST60_ET200SP_CM_4xIO_Link_3[30] := HwInputs.ST60_ET200SP_CM_4xIO_Link_3[30];
	PlcInputs.ST60_ET200SP_CM_4xIO_Link_3[31] := HwInputs.ST60_ET200SP_CM_4xIO_Link_3[31];
	PlcInputs.ST60_ET200SP_AI_4xI_2_4_wire_ST_1[0] := HwInputs.ST60_ET200SP_AI_4xI_2_4_wire_ST_1[0];
	PlcInputs.ST60_ET200SP_AI_4xI_2_4_wire_ST_1[1] := HwInputs.ST60_ET200SP_AI_4xI_2_4_wire_ST_1[1];
	PlcInputs.ST60_ET200SP_AI_4xI_2_4_wire_ST_1[2] := HwInputs.ST60_ET200SP_AI_4xI_2_4_wire_ST_1[2];
	PlcInputs.ST60_ET200SP_AI_4xI_2_4_wire_ST_1[3] := HwInputs.ST60_ET200SP_AI_4xI_2_4_wire_ST_1[3];
	PlcInputs.ST60_ET200SP_AI_4xI_2_4_wire_ST_1[4] := HwInputs.ST60_ET200SP_AI_4xI_2_4_wire_ST_1[4];
	PlcInputs.ST60_ET200SP_AI_4xI_2_4_wire_ST_1[5] := HwInputs.ST60_ET200SP_AI_4xI_2_4_wire_ST_1[5];
	PlcInputs.ST60_ET200SP_AI_4xI_2_4_wire_ST_1[6] := HwInputs.ST60_ET200SP_AI_4xI_2_4_wire_ST_1[6];
	PlcInputs.ST60_ET200SP_AI_4xI_2_4_wire_ST_1[7] := HwInputs.ST60_ET200SP_AI_4xI_2_4_wire_ST_1[7];
	PlcInputs.ST60_ET200SP_DI_16x24VDC_ST_1 := HwInputs.ST60_ET200SP_DI_16x24VDC_ST_1;
	PlcInputs.ST60_ET200SP_DI_16x24VDC_ST_2 := HwInputs.ST60_ET200SP_DI_16x24VDC_ST_2;
	PlcInputs.ST60_ET200SP_DI_8x24VDC_ST_4 := HwInputs.ST60_ET200SP_DI_8x24VDC_ST_4;
	PlcInputs.ST60_ET200SP_DI_8x24VDC_ST_3 := HwInputs.ST60_ET200SP_DI_8x24VDC_ST_3;
	PlcInputs.ST60_6_DM260_Acquisition_Status[0] := HwInputs.ST60_6_DM260_Acquisition_Status[0];
	PlcInputs.ST60_6_DM260_Acquisition_Status[1] := HwInputs.ST60_6_DM260_Acquisition_Status[1];
	PlcInputs.ST60_6_DM260_Acquisition_Status[2] := HwInputs.ST60_6_DM260_Acquisition_Status[2];
	PlcInputs.ST60_6_DM260_Results_Status := HwInputs.ST60_6_DM260_Results_Status;
	PlcInputs.ST60_6_DM260_Soft_Event_Control := HwInputs.ST60_6_DM260_Soft_Event_Control;
	PlcInputs.ST60_6_DM260_Result_Data_64_bytes[0] := HwInputs.ST60_6_DM260_Result_Data_64_bytes[0];
	PlcInputs.ST60_6_DM260_Result_Data_64_bytes[1] := HwInputs.ST60_6_DM260_Result_Data_64_bytes[1];
	PlcInputs.ST60_6_DM260_Result_Data_64_bytes[2] := HwInputs.ST60_6_DM260_Result_Data_64_bytes[2];
	PlcInputs.ST60_6_DM260_Result_Data_64_bytes[3] := HwInputs.ST60_6_DM260_Result_Data_64_bytes[3];
	PlcInputs.ST60_6_DM260_Result_Data_64_bytes[4] := HwInputs.ST60_6_DM260_Result_Data_64_bytes[4];
	PlcInputs.ST60_6_DM260_Result_Data_64_bytes[5] := HwInputs.ST60_6_DM260_Result_Data_64_bytes[5];
	PlcInputs.ST60_6_DM260_Result_Data_64_bytes[6] := HwInputs.ST60_6_DM260_Result_Data_64_bytes[6];
	PlcInputs.ST60_6_DM260_Result_Data_64_bytes[7] := HwInputs.ST60_6_DM260_Result_Data_64_bytes[7];
	PlcInputs.ST60_6_DM260_Result_Data_64_bytes[8] := HwInputs.ST60_6_DM260_Result_Data_64_bytes[8];
	PlcInputs.ST60_6_DM260_Result_Data_64_bytes[9] := HwInputs.ST60_6_DM260_Result_Data_64_bytes[9];
	PlcInputs.ST60_6_DM260_Result_Data_64_bytes[10] := HwInputs.ST60_6_DM260_Result_Data_64_bytes[10];
	PlcInputs.ST60_6_DM260_Result_Data_64_bytes[11] := HwInputs.ST60_6_DM260_Result_Data_64_bytes[11];
	PlcInputs.ST60_6_DM260_Result_Data_64_bytes[12] := HwInputs.ST60_6_DM260_Result_Data_64_bytes[12];
	PlcInputs.ST60_6_DM260_Result_Data_64_bytes[13] := HwInputs.ST60_6_DM260_Result_Data_64_bytes[13];
	PlcInputs.ST60_6_DM260_Result_Data_64_bytes[14] := HwInputs.ST60_6_DM260_Result_Data_64_bytes[14];
	PlcInputs.ST60_6_DM260_Result_Data_64_bytes[15] := HwInputs.ST60_6_DM260_Result_Data_64_bytes[15];
	PlcInputs.ST60_6_DM260_Result_Data_64_bytes[16] := HwInputs.ST60_6_DM260_Result_Data_64_bytes[16];
	PlcInputs.ST60_6_DM260_Result_Data_64_bytes[17] := HwInputs.ST60_6_DM260_Result_Data_64_bytes[17];
	PlcInputs.ST60_6_DM260_Result_Data_64_bytes[18] := HwInputs.ST60_6_DM260_Result_Data_64_bytes[18];
	PlcInputs.ST60_6_DM260_Result_Data_64_bytes[19] := HwInputs.ST60_6_DM260_Result_Data_64_bytes[19];
	PlcInputs.ST60_6_DM260_Result_Data_64_bytes[20] := HwInputs.ST60_6_DM260_Result_Data_64_bytes[20];
	PlcInputs.ST60_6_DM260_Result_Data_64_bytes[21] := HwInputs.ST60_6_DM260_Result_Data_64_bytes[21];
	PlcInputs.ST60_6_DM260_Result_Data_64_bytes[22] := HwInputs.ST60_6_DM260_Result_Data_64_bytes[22];
	PlcInputs.ST60_6_DM260_Result_Data_64_bytes[23] := HwInputs.ST60_6_DM260_Result_Data_64_bytes[23];
	PlcInputs.ST60_6_DM260_Result_Data_64_bytes[24] := HwInputs.ST60_6_DM260_Result_Data_64_bytes[24];
	PlcInputs.ST60_6_DM260_Result_Data_64_bytes[25] := HwInputs.ST60_6_DM260_Result_Data_64_bytes[25];
	PlcInputs.ST60_6_DM260_Result_Data_64_bytes[26] := HwInputs.ST60_6_DM260_Result_Data_64_bytes[26];
	PlcInputs.ST60_6_DM260_Result_Data_64_bytes[27] := HwInputs.ST60_6_DM260_Result_Data_64_bytes[27];
	PlcInputs.ST60_6_DM260_Result_Data_64_bytes[28] := HwInputs.ST60_6_DM260_Result_Data_64_bytes[28];
	PlcInputs.ST60_6_DM260_Result_Data_64_bytes[29] := HwInputs.ST60_6_DM260_Result_Data_64_bytes[29];
	PlcInputs.ST60_6_DM260_Result_Data_64_bytes[30] := HwInputs.ST60_6_DM260_Result_Data_64_bytes[30];
	PlcInputs.ST60_6_DM260_Result_Data_64_bytes[31] := HwInputs.ST60_6_DM260_Result_Data_64_bytes[31];
	PlcInputs.ST60_6_DM260_Result_Data_64_bytes[32] := HwInputs.ST60_6_DM260_Result_Data_64_bytes[32];
	PlcInputs.ST60_6_DM260_Result_Data_64_bytes[33] := HwInputs.ST60_6_DM260_Result_Data_64_bytes[33];
	PlcInputs.ST60_6_DM260_Result_Data_64_bytes[34] := HwInputs.ST60_6_DM260_Result_Data_64_bytes[34];
	PlcInputs.ST60_6_DM260_Result_Data_64_bytes[35] := HwInputs.ST60_6_DM260_Result_Data_64_bytes[35];
	PlcInputs.ST60_6_DM260_Result_Data_64_bytes[36] := HwInputs.ST60_6_DM260_Result_Data_64_bytes[36];
	PlcInputs.ST60_6_DM260_Result_Data_64_bytes[37] := HwInputs.ST60_6_DM260_Result_Data_64_bytes[37];
	PlcInputs.ST60_6_DM260_Result_Data_64_bytes[38] := HwInputs.ST60_6_DM260_Result_Data_64_bytes[38];
	PlcInputs.ST60_6_DM260_Result_Data_64_bytes[39] := HwInputs.ST60_6_DM260_Result_Data_64_bytes[39];
	PlcInputs.ST60_6_DM260_Result_Data_64_bytes[40] := HwInputs.ST60_6_DM260_Result_Data_64_bytes[40];
	PlcInputs.ST60_6_DM260_Result_Data_64_bytes[41] := HwInputs.ST60_6_DM260_Result_Data_64_bytes[41];
	PlcInputs.ST60_6_DM260_Result_Data_64_bytes[42] := HwInputs.ST60_6_DM260_Result_Data_64_bytes[42];
	PlcInputs.ST60_6_DM260_Result_Data_64_bytes[43] := HwInputs.ST60_6_DM260_Result_Data_64_bytes[43];
	PlcInputs.ST60_6_DM260_Result_Data_64_bytes[44] := HwInputs.ST60_6_DM260_Result_Data_64_bytes[44];
	PlcInputs.ST60_6_DM260_Result_Data_64_bytes[45] := HwInputs.ST60_6_DM260_Result_Data_64_bytes[45];
	PlcInputs.ST60_6_DM260_Result_Data_64_bytes[46] := HwInputs.ST60_6_DM260_Result_Data_64_bytes[46];
	PlcInputs.ST60_6_DM260_Result_Data_64_bytes[47] := HwInputs.ST60_6_DM260_Result_Data_64_bytes[47];
	PlcInputs.ST60_6_DM260_Result_Data_64_bytes[48] := HwInputs.ST60_6_DM260_Result_Data_64_bytes[48];
	PlcInputs.ST60_6_DM260_Result_Data_64_bytes[49] := HwInputs.ST60_6_DM260_Result_Data_64_bytes[49];
	PlcInputs.ST60_6_DM260_Result_Data_64_bytes[50] := HwInputs.ST60_6_DM260_Result_Data_64_bytes[50];
	PlcInputs.ST60_6_DM260_Result_Data_64_bytes[51] := HwInputs.ST60_6_DM260_Result_Data_64_bytes[51];
	PlcInputs.ST60_6_DM260_Result_Data_64_bytes[52] := HwInputs.ST60_6_DM260_Result_Data_64_bytes[52];
	PlcInputs.ST60_6_DM260_Result_Data_64_bytes[53] := HwInputs.ST60_6_DM260_Result_Data_64_bytes[53];
	PlcInputs.ST60_6_DM260_Result_Data_64_bytes[54] := HwInputs.ST60_6_DM260_Result_Data_64_bytes[54];
	PlcInputs.ST60_6_DM260_Result_Data_64_bytes[55] := HwInputs.ST60_6_DM260_Result_Data_64_bytes[55];
	PlcInputs.ST60_6_DM260_Result_Data_64_bytes[56] := HwInputs.ST60_6_DM260_Result_Data_64_bytes[56];
	PlcInputs.ST60_6_DM260_Result_Data_64_bytes[57] := HwInputs.ST60_6_DM260_Result_Data_64_bytes[57];
	PlcInputs.ST60_6_DM260_Result_Data_64_bytes[58] := HwInputs.ST60_6_DM260_Result_Data_64_bytes[58];
	PlcInputs.ST60_6_DM260_Result_Data_64_bytes[59] := HwInputs.ST60_6_DM260_Result_Data_64_bytes[59];
	PlcInputs.ST60_6_DM260_Result_Data_64_bytes[60] := HwInputs.ST60_6_DM260_Result_Data_64_bytes[60];
	PlcInputs.ST60_6_DM260_Result_Data_64_bytes[61] := HwInputs.ST60_6_DM260_Result_Data_64_bytes[61];
	PlcInputs.ST60_6_DM260_Result_Data_64_bytes[62] := HwInputs.ST60_6_DM260_Result_Data_64_bytes[62];
	PlcInputs.ST60_6_DM260_Result_Data_64_bytes[63] := HwInputs.ST60_6_DM260_Result_Data_64_bytes[63];
	PlcInputs.ST60_6_DM260_Result_Data_64_bytes[64] := HwInputs.ST60_6_DM260_Result_Data_64_bytes[64];
	PlcInputs.ST60_6_DM260_Result_Data_64_bytes[65] := HwInputs.ST60_6_DM260_Result_Data_64_bytes[65];
	PlcInputs.ST60_6_DM260_Result_Data_64_bytes[66] := HwInputs.ST60_6_DM260_Result_Data_64_bytes[66];
	PlcInputs.ST60_6_DM260_Result_Data_64_bytes[67] := HwInputs.ST60_6_DM260_Result_Data_64_bytes[67];
	PlcInputs.ST60_6_DM260_Result_Data_64_bytes[68] := HwInputs.ST60_6_DM260_Result_Data_64_bytes[68];
	PlcInputs.ST60_6_DM260_Result_Data_64_bytes[69] := HwInputs.ST60_6_DM260_Result_Data_64_bytes[69];
	PlcInputs.ST60_6_DM260_Result_Data_64_bytes[70] := HwInputs.ST60_6_DM260_Result_Data_64_bytes[70];
	PlcInputs.ST60_6_DM260_Result_Data_64_bytes[71] := HwInputs.ST60_6_DM260_Result_Data_64_bytes[71];
	PlcInputs.ST60_3_DM260_Acquisition_Status[0] := HwInputs.ST60_3_DM260_Acquisition_Status[0];
	PlcInputs.ST60_3_DM260_Acquisition_Status[1] := HwInputs.ST60_3_DM260_Acquisition_Status[1];
	PlcInputs.ST60_3_DM260_Acquisition_Status[2] := HwInputs.ST60_3_DM260_Acquisition_Status[2];
	PlcInputs.ST60_3_DM260_Results_Status := HwInputs.ST60_3_DM260_Results_Status;
	PlcInputs.ST60_3_DM260_Soft_Event_Control := HwInputs.ST60_3_DM260_Soft_Event_Control;
	PlcInputs.ST60_3_DM260_Result_Data_64_bytes[0] := HwInputs.ST60_3_DM260_Result_Data_64_bytes[0];
	PlcInputs.ST60_3_DM260_Result_Data_64_bytes[1] := HwInputs.ST60_3_DM260_Result_Data_64_bytes[1];
	PlcInputs.ST60_3_DM260_Result_Data_64_bytes[2] := HwInputs.ST60_3_DM260_Result_Data_64_bytes[2];
	PlcInputs.ST60_3_DM260_Result_Data_64_bytes[3] := HwInputs.ST60_3_DM260_Result_Data_64_bytes[3];
	PlcInputs.ST60_3_DM260_Result_Data_64_bytes[4] := HwInputs.ST60_3_DM260_Result_Data_64_bytes[4];
	PlcInputs.ST60_3_DM260_Result_Data_64_bytes[5] := HwInputs.ST60_3_DM260_Result_Data_64_bytes[5];
	PlcInputs.ST60_3_DM260_Result_Data_64_bytes[6] := HwInputs.ST60_3_DM260_Result_Data_64_bytes[6];
	PlcInputs.ST60_3_DM260_Result_Data_64_bytes[7] := HwInputs.ST60_3_DM260_Result_Data_64_bytes[7];
	PlcInputs.ST60_3_DM260_Result_Data_64_bytes[8] := HwInputs.ST60_3_DM260_Result_Data_64_bytes[8];
	PlcInputs.ST60_3_DM260_Result_Data_64_bytes[9] := HwInputs.ST60_3_DM260_Result_Data_64_bytes[9];
	PlcInputs.ST60_3_DM260_Result_Data_64_bytes[10] := HwInputs.ST60_3_DM260_Result_Data_64_bytes[10];
	PlcInputs.ST60_3_DM260_Result_Data_64_bytes[11] := HwInputs.ST60_3_DM260_Result_Data_64_bytes[11];
	PlcInputs.ST60_3_DM260_Result_Data_64_bytes[12] := HwInputs.ST60_3_DM260_Result_Data_64_bytes[12];
	PlcInputs.ST60_3_DM260_Result_Data_64_bytes[13] := HwInputs.ST60_3_DM260_Result_Data_64_bytes[13];
	PlcInputs.ST60_3_DM260_Result_Data_64_bytes[14] := HwInputs.ST60_3_DM260_Result_Data_64_bytes[14];
	PlcInputs.ST60_3_DM260_Result_Data_64_bytes[15] := HwInputs.ST60_3_DM260_Result_Data_64_bytes[15];
	PlcInputs.ST60_3_DM260_Result_Data_64_bytes[16] := HwInputs.ST60_3_DM260_Result_Data_64_bytes[16];
	PlcInputs.ST60_3_DM260_Result_Data_64_bytes[17] := HwInputs.ST60_3_DM260_Result_Data_64_bytes[17];
	PlcInputs.ST60_3_DM260_Result_Data_64_bytes[18] := HwInputs.ST60_3_DM260_Result_Data_64_bytes[18];
	PlcInputs.ST60_3_DM260_Result_Data_64_bytes[19] := HwInputs.ST60_3_DM260_Result_Data_64_bytes[19];
	PlcInputs.ST60_3_DM260_Result_Data_64_bytes[20] := HwInputs.ST60_3_DM260_Result_Data_64_bytes[20];
	PlcInputs.ST60_3_DM260_Result_Data_64_bytes[21] := HwInputs.ST60_3_DM260_Result_Data_64_bytes[21];
	PlcInputs.ST60_3_DM260_Result_Data_64_bytes[22] := HwInputs.ST60_3_DM260_Result_Data_64_bytes[22];
	PlcInputs.ST60_3_DM260_Result_Data_64_bytes[23] := HwInputs.ST60_3_DM260_Result_Data_64_bytes[23];
	PlcInputs.ST60_3_DM260_Result_Data_64_bytes[24] := HwInputs.ST60_3_DM260_Result_Data_64_bytes[24];
	PlcInputs.ST60_3_DM260_Result_Data_64_bytes[25] := HwInputs.ST60_3_DM260_Result_Data_64_bytes[25];
	PlcInputs.ST60_3_DM260_Result_Data_64_bytes[26] := HwInputs.ST60_3_DM260_Result_Data_64_bytes[26];
	PlcInputs.ST60_3_DM260_Result_Data_64_bytes[27] := HwInputs.ST60_3_DM260_Result_Data_64_bytes[27];
	PlcInputs.ST60_3_DM260_Result_Data_64_bytes[28] := HwInputs.ST60_3_DM260_Result_Data_64_bytes[28];
	PlcInputs.ST60_3_DM260_Result_Data_64_bytes[29] := HwInputs.ST60_3_DM260_Result_Data_64_bytes[29];
	PlcInputs.ST60_3_DM260_Result_Data_64_bytes[30] := HwInputs.ST60_3_DM260_Result_Data_64_bytes[30];
	PlcInputs.ST60_3_DM260_Result_Data_64_bytes[31] := HwInputs.ST60_3_DM260_Result_Data_64_bytes[31];
	PlcInputs.ST60_3_DM260_Result_Data_64_bytes[32] := HwInputs.ST60_3_DM260_Result_Data_64_bytes[32];
	PlcInputs.ST60_3_DM260_Result_Data_64_bytes[33] := HwInputs.ST60_3_DM260_Result_Data_64_bytes[33];
	PlcInputs.ST60_3_DM260_Result_Data_64_bytes[34] := HwInputs.ST60_3_DM260_Result_Data_64_bytes[34];
	PlcInputs.ST60_3_DM260_Result_Data_64_bytes[35] := HwInputs.ST60_3_DM260_Result_Data_64_bytes[35];
	PlcInputs.ST60_3_DM260_Result_Data_64_bytes[36] := HwInputs.ST60_3_DM260_Result_Data_64_bytes[36];
	PlcInputs.ST60_3_DM260_Result_Data_64_bytes[37] := HwInputs.ST60_3_DM260_Result_Data_64_bytes[37];
	PlcInputs.ST60_3_DM260_Result_Data_64_bytes[38] := HwInputs.ST60_3_DM260_Result_Data_64_bytes[38];
	PlcInputs.ST60_3_DM260_Result_Data_64_bytes[39] := HwInputs.ST60_3_DM260_Result_Data_64_bytes[39];
	PlcInputs.ST60_3_DM260_Result_Data_64_bytes[40] := HwInputs.ST60_3_DM260_Result_Data_64_bytes[40];
	PlcInputs.ST60_3_DM260_Result_Data_64_bytes[41] := HwInputs.ST60_3_DM260_Result_Data_64_bytes[41];
	PlcInputs.ST60_3_DM260_Result_Data_64_bytes[42] := HwInputs.ST60_3_DM260_Result_Data_64_bytes[42];
	PlcInputs.ST60_3_DM260_Result_Data_64_bytes[43] := HwInputs.ST60_3_DM260_Result_Data_64_bytes[43];
	PlcInputs.ST60_3_DM260_Result_Data_64_bytes[44] := HwInputs.ST60_3_DM260_Result_Data_64_bytes[44];
	PlcInputs.ST60_3_DM260_Result_Data_64_bytes[45] := HwInputs.ST60_3_DM260_Result_Data_64_bytes[45];
	PlcInputs.ST60_3_DM260_Result_Data_64_bytes[46] := HwInputs.ST60_3_DM260_Result_Data_64_bytes[46];
	PlcInputs.ST60_3_DM260_Result_Data_64_bytes[47] := HwInputs.ST60_3_DM260_Result_Data_64_bytes[47];
	PlcInputs.ST60_3_DM260_Result_Data_64_bytes[48] := HwInputs.ST60_3_DM260_Result_Data_64_bytes[48];
	PlcInputs.ST60_3_DM260_Result_Data_64_bytes[49] := HwInputs.ST60_3_DM260_Result_Data_64_bytes[49];
	PlcInputs.ST60_3_DM260_Result_Data_64_bytes[50] := HwInputs.ST60_3_DM260_Result_Data_64_bytes[50];
	PlcInputs.ST60_3_DM260_Result_Data_64_bytes[51] := HwInputs.ST60_3_DM260_Result_Data_64_bytes[51];
	PlcInputs.ST60_3_DM260_Result_Data_64_bytes[52] := HwInputs.ST60_3_DM260_Result_Data_64_bytes[52];
	PlcInputs.ST60_3_DM260_Result_Data_64_bytes[53] := HwInputs.ST60_3_DM260_Result_Data_64_bytes[53];
	PlcInputs.ST60_3_DM260_Result_Data_64_bytes[54] := HwInputs.ST60_3_DM260_Result_Data_64_bytes[54];
	PlcInputs.ST60_3_DM260_Result_Data_64_bytes[55] := HwInputs.ST60_3_DM260_Result_Data_64_bytes[55];
	PlcInputs.ST60_3_DM260_Result_Data_64_bytes[56] := HwInputs.ST60_3_DM260_Result_Data_64_bytes[56];
	PlcInputs.ST60_3_DM260_Result_Data_64_bytes[57] := HwInputs.ST60_3_DM260_Result_Data_64_bytes[57];
	PlcInputs.ST60_3_DM260_Result_Data_64_bytes[58] := HwInputs.ST60_3_DM260_Result_Data_64_bytes[58];
	PlcInputs.ST60_3_DM260_Result_Data_64_bytes[59] := HwInputs.ST60_3_DM260_Result_Data_64_bytes[59];
	PlcInputs.ST60_3_DM260_Result_Data_64_bytes[60] := HwInputs.ST60_3_DM260_Result_Data_64_bytes[60];
	PlcInputs.ST60_3_DM260_Result_Data_64_bytes[61] := HwInputs.ST60_3_DM260_Result_Data_64_bytes[61];
	PlcInputs.ST60_3_DM260_Result_Data_64_bytes[62] := HwInputs.ST60_3_DM260_Result_Data_64_bytes[62];
	PlcInputs.ST60_3_DM260_Result_Data_64_bytes[63] := HwInputs.ST60_3_DM260_Result_Data_64_bytes[63];
	PlcInputs.ST60_3_DM260_Result_Data_64_bytes[64] := HwInputs.ST60_3_DM260_Result_Data_64_bytes[64];
	PlcInputs.ST60_3_DM260_Result_Data_64_bytes[65] := HwInputs.ST60_3_DM260_Result_Data_64_bytes[65];
	PlcInputs.ST60_3_DM260_Result_Data_64_bytes[66] := HwInputs.ST60_3_DM260_Result_Data_64_bytes[66];
	PlcInputs.ST60_3_DM260_Result_Data_64_bytes[67] := HwInputs.ST60_3_DM260_Result_Data_64_bytes[67];
	PlcInputs.ST60_3_DM260_Result_Data_64_bytes[68] := HwInputs.ST60_3_DM260_Result_Data_64_bytes[68];
	PlcInputs.ST60_3_DM260_Result_Data_64_bytes[69] := HwInputs.ST60_3_DM260_Result_Data_64_bytes[69];
	PlcInputs.ST60_3_DM260_Result_Data_64_bytes[70] := HwInputs.ST60_3_DM260_Result_Data_64_bytes[70];
	PlcInputs.ST60_3_DM260_Result_Data_64_bytes[71] := HwInputs.ST60_3_DM260_Result_Data_64_bytes[71];
	PlcInputs.ST60_4_DM260_Acquisition_Status[0] := HwInputs.ST60_4_DM260_Acquisition_Status[0];
	PlcInputs.ST60_4_DM260_Acquisition_Status[1] := HwInputs.ST60_4_DM260_Acquisition_Status[1];
	PlcInputs.ST60_4_DM260_Acquisition_Status[2] := HwInputs.ST60_4_DM260_Acquisition_Status[2];
	PlcInputs.ST60_4_DM260_Results_Status := HwInputs.ST60_4_DM260_Results_Status;
	PlcInputs.ST60_4_DM260_Soft_Event_Control := HwInputs.ST60_4_DM260_Soft_Event_Control;
	PlcInputs.ST60_4_DM260_Result_Data_64_bytes[0] := HwInputs.ST60_4_DM260_Result_Data_64_bytes[0];
	PlcInputs.ST60_4_DM260_Result_Data_64_bytes[1] := HwInputs.ST60_4_DM260_Result_Data_64_bytes[1];
	PlcInputs.ST60_4_DM260_Result_Data_64_bytes[2] := HwInputs.ST60_4_DM260_Result_Data_64_bytes[2];
	PlcInputs.ST60_4_DM260_Result_Data_64_bytes[3] := HwInputs.ST60_4_DM260_Result_Data_64_bytes[3];
	PlcInputs.ST60_4_DM260_Result_Data_64_bytes[4] := HwInputs.ST60_4_DM260_Result_Data_64_bytes[4];
	PlcInputs.ST60_4_DM260_Result_Data_64_bytes[5] := HwInputs.ST60_4_DM260_Result_Data_64_bytes[5];
	PlcInputs.ST60_4_DM260_Result_Data_64_bytes[6] := HwInputs.ST60_4_DM260_Result_Data_64_bytes[6];
	PlcInputs.ST60_4_DM260_Result_Data_64_bytes[7] := HwInputs.ST60_4_DM260_Result_Data_64_bytes[7];
	PlcInputs.ST60_4_DM260_Result_Data_64_bytes[8] := HwInputs.ST60_4_DM260_Result_Data_64_bytes[8];
	PlcInputs.ST60_4_DM260_Result_Data_64_bytes[9] := HwInputs.ST60_4_DM260_Result_Data_64_bytes[9];
	PlcInputs.ST60_4_DM260_Result_Data_64_bytes[10] := HwInputs.ST60_4_DM260_Result_Data_64_bytes[10];
	PlcInputs.ST60_4_DM260_Result_Data_64_bytes[11] := HwInputs.ST60_4_DM260_Result_Data_64_bytes[11];
	PlcInputs.ST60_4_DM260_Result_Data_64_bytes[12] := HwInputs.ST60_4_DM260_Result_Data_64_bytes[12];
	PlcInputs.ST60_4_DM260_Result_Data_64_bytes[13] := HwInputs.ST60_4_DM260_Result_Data_64_bytes[13];
	PlcInputs.ST60_4_DM260_Result_Data_64_bytes[14] := HwInputs.ST60_4_DM260_Result_Data_64_bytes[14];
	PlcInputs.ST60_4_DM260_Result_Data_64_bytes[15] := HwInputs.ST60_4_DM260_Result_Data_64_bytes[15];
	PlcInputs.ST60_4_DM260_Result_Data_64_bytes[16] := HwInputs.ST60_4_DM260_Result_Data_64_bytes[16];
	PlcInputs.ST60_4_DM260_Result_Data_64_bytes[17] := HwInputs.ST60_4_DM260_Result_Data_64_bytes[17];
	PlcInputs.ST60_4_DM260_Result_Data_64_bytes[18] := HwInputs.ST60_4_DM260_Result_Data_64_bytes[18];
	PlcInputs.ST60_4_DM260_Result_Data_64_bytes[19] := HwInputs.ST60_4_DM260_Result_Data_64_bytes[19];
	PlcInputs.ST60_4_DM260_Result_Data_64_bytes[20] := HwInputs.ST60_4_DM260_Result_Data_64_bytes[20];
	PlcInputs.ST60_4_DM260_Result_Data_64_bytes[21] := HwInputs.ST60_4_DM260_Result_Data_64_bytes[21];
	PlcInputs.ST60_4_DM260_Result_Data_64_bytes[22] := HwInputs.ST60_4_DM260_Result_Data_64_bytes[22];
	PlcInputs.ST60_4_DM260_Result_Data_64_bytes[23] := HwInputs.ST60_4_DM260_Result_Data_64_bytes[23];
	PlcInputs.ST60_4_DM260_Result_Data_64_bytes[24] := HwInputs.ST60_4_DM260_Result_Data_64_bytes[24];
	PlcInputs.ST60_4_DM260_Result_Data_64_bytes[25] := HwInputs.ST60_4_DM260_Result_Data_64_bytes[25];
	PlcInputs.ST60_4_DM260_Result_Data_64_bytes[26] := HwInputs.ST60_4_DM260_Result_Data_64_bytes[26];
	PlcInputs.ST60_4_DM260_Result_Data_64_bytes[27] := HwInputs.ST60_4_DM260_Result_Data_64_bytes[27];
	PlcInputs.ST60_4_DM260_Result_Data_64_bytes[28] := HwInputs.ST60_4_DM260_Result_Data_64_bytes[28];
	PlcInputs.ST60_4_DM260_Result_Data_64_bytes[29] := HwInputs.ST60_4_DM260_Result_Data_64_bytes[29];
	PlcInputs.ST60_4_DM260_Result_Data_64_bytes[30] := HwInputs.ST60_4_DM260_Result_Data_64_bytes[30];
	PlcInputs.ST60_4_DM260_Result_Data_64_bytes[31] := HwInputs.ST60_4_DM260_Result_Data_64_bytes[31];
	PlcInputs.ST60_4_DM260_Result_Data_64_bytes[32] := HwInputs.ST60_4_DM260_Result_Data_64_bytes[32];
	PlcInputs.ST60_4_DM260_Result_Data_64_bytes[33] := HwInputs.ST60_4_DM260_Result_Data_64_bytes[33];
	PlcInputs.ST60_4_DM260_Result_Data_64_bytes[34] := HwInputs.ST60_4_DM260_Result_Data_64_bytes[34];
	PlcInputs.ST60_4_DM260_Result_Data_64_bytes[35] := HwInputs.ST60_4_DM260_Result_Data_64_bytes[35];
	PlcInputs.ST60_4_DM260_Result_Data_64_bytes[36] := HwInputs.ST60_4_DM260_Result_Data_64_bytes[36];
	PlcInputs.ST60_4_DM260_Result_Data_64_bytes[37] := HwInputs.ST60_4_DM260_Result_Data_64_bytes[37];
	PlcInputs.ST60_4_DM260_Result_Data_64_bytes[38] := HwInputs.ST60_4_DM260_Result_Data_64_bytes[38];
	PlcInputs.ST60_4_DM260_Result_Data_64_bytes[39] := HwInputs.ST60_4_DM260_Result_Data_64_bytes[39];
	PlcInputs.ST60_4_DM260_Result_Data_64_bytes[40] := HwInputs.ST60_4_DM260_Result_Data_64_bytes[40];
	PlcInputs.ST60_4_DM260_Result_Data_64_bytes[41] := HwInputs.ST60_4_DM260_Result_Data_64_bytes[41];
	PlcInputs.ST60_4_DM260_Result_Data_64_bytes[42] := HwInputs.ST60_4_DM260_Result_Data_64_bytes[42];
	PlcInputs.ST60_4_DM260_Result_Data_64_bytes[43] := HwInputs.ST60_4_DM260_Result_Data_64_bytes[43];
	PlcInputs.ST60_4_DM260_Result_Data_64_bytes[44] := HwInputs.ST60_4_DM260_Result_Data_64_bytes[44];
	PlcInputs.ST60_4_DM260_Result_Data_64_bytes[45] := HwInputs.ST60_4_DM260_Result_Data_64_bytes[45];
	PlcInputs.ST60_4_DM260_Result_Data_64_bytes[46] := HwInputs.ST60_4_DM260_Result_Data_64_bytes[46];
	PlcInputs.ST60_4_DM260_Result_Data_64_bytes[47] := HwInputs.ST60_4_DM260_Result_Data_64_bytes[47];
	PlcInputs.ST60_4_DM260_Result_Data_64_bytes[48] := HwInputs.ST60_4_DM260_Result_Data_64_bytes[48];
	PlcInputs.ST60_4_DM260_Result_Data_64_bytes[49] := HwInputs.ST60_4_DM260_Result_Data_64_bytes[49];
	PlcInputs.ST60_4_DM260_Result_Data_64_bytes[50] := HwInputs.ST60_4_DM260_Result_Data_64_bytes[50];
	PlcInputs.ST60_4_DM260_Result_Data_64_bytes[51] := HwInputs.ST60_4_DM260_Result_Data_64_bytes[51];
	PlcInputs.ST60_4_DM260_Result_Data_64_bytes[52] := HwInputs.ST60_4_DM260_Result_Data_64_bytes[52];
	PlcInputs.ST60_4_DM260_Result_Data_64_bytes[53] := HwInputs.ST60_4_DM260_Result_Data_64_bytes[53];
	PlcInputs.ST60_4_DM260_Result_Data_64_bytes[54] := HwInputs.ST60_4_DM260_Result_Data_64_bytes[54];
	PlcInputs.ST60_4_DM260_Result_Data_64_bytes[55] := HwInputs.ST60_4_DM260_Result_Data_64_bytes[55];
	PlcInputs.ST60_4_DM260_Result_Data_64_bytes[56] := HwInputs.ST60_4_DM260_Result_Data_64_bytes[56];
	PlcInputs.ST60_4_DM260_Result_Data_64_bytes[57] := HwInputs.ST60_4_DM260_Result_Data_64_bytes[57];
	PlcInputs.ST60_4_DM260_Result_Data_64_bytes[58] := HwInputs.ST60_4_DM260_Result_Data_64_bytes[58];
	PlcInputs.ST60_4_DM260_Result_Data_64_bytes[59] := HwInputs.ST60_4_DM260_Result_Data_64_bytes[59];
	PlcInputs.ST60_4_DM260_Result_Data_64_bytes[60] := HwInputs.ST60_4_DM260_Result_Data_64_bytes[60];
	PlcInputs.ST60_4_DM260_Result_Data_64_bytes[61] := HwInputs.ST60_4_DM260_Result_Data_64_bytes[61];
	PlcInputs.ST60_4_DM260_Result_Data_64_bytes[62] := HwInputs.ST60_4_DM260_Result_Data_64_bytes[62];
	PlcInputs.ST60_4_DM260_Result_Data_64_bytes[63] := HwInputs.ST60_4_DM260_Result_Data_64_bytes[63];
	PlcInputs.ST60_4_DM260_Result_Data_64_bytes[64] := HwInputs.ST60_4_DM260_Result_Data_64_bytes[64];
	PlcInputs.ST60_4_DM260_Result_Data_64_bytes[65] := HwInputs.ST60_4_DM260_Result_Data_64_bytes[65];
	PlcInputs.ST60_4_DM260_Result_Data_64_bytes[66] := HwInputs.ST60_4_DM260_Result_Data_64_bytes[66];
	PlcInputs.ST60_4_DM260_Result_Data_64_bytes[67] := HwInputs.ST60_4_DM260_Result_Data_64_bytes[67];
	PlcInputs.ST60_4_DM260_Result_Data_64_bytes[68] := HwInputs.ST60_4_DM260_Result_Data_64_bytes[68];
	PlcInputs.ST60_4_DM260_Result_Data_64_bytes[69] := HwInputs.ST60_4_DM260_Result_Data_64_bytes[69];
	PlcInputs.ST60_4_DM260_Result_Data_64_bytes[70] := HwInputs.ST60_4_DM260_Result_Data_64_bytes[70];
	PlcInputs.ST60_4_DM260_Result_Data_64_bytes[71] := HwInputs.ST60_4_DM260_Result_Data_64_bytes[71];
	PlcInputs.ST60_5_DM260_Acquisition_Status[0] := HwInputs.ST60_5_DM260_Acquisition_Status[0];
	PlcInputs.ST60_5_DM260_Acquisition_Status[1] := HwInputs.ST60_5_DM260_Acquisition_Status[1];
	PlcInputs.ST60_5_DM260_Acquisition_Status[2] := HwInputs.ST60_5_DM260_Acquisition_Status[2];
	PlcInputs.ST60_5_DM260_Results_Status := HwInputs.ST60_5_DM260_Results_Status;
	PlcInputs.ST60_5_DM260_Soft_Event_Control := HwInputs.ST60_5_DM260_Soft_Event_Control;
	PlcInputs.ST60_5_DM260_Result_Data_64_bytes[0] := HwInputs.ST60_5_DM260_Result_Data_64_bytes[0];
	PlcInputs.ST60_5_DM260_Result_Data_64_bytes[1] := HwInputs.ST60_5_DM260_Result_Data_64_bytes[1];
	PlcInputs.ST60_5_DM260_Result_Data_64_bytes[2] := HwInputs.ST60_5_DM260_Result_Data_64_bytes[2];
	PlcInputs.ST60_5_DM260_Result_Data_64_bytes[3] := HwInputs.ST60_5_DM260_Result_Data_64_bytes[3];
	PlcInputs.ST60_5_DM260_Result_Data_64_bytes[4] := HwInputs.ST60_5_DM260_Result_Data_64_bytes[4];
	PlcInputs.ST60_5_DM260_Result_Data_64_bytes[5] := HwInputs.ST60_5_DM260_Result_Data_64_bytes[5];
	PlcInputs.ST60_5_DM260_Result_Data_64_bytes[6] := HwInputs.ST60_5_DM260_Result_Data_64_bytes[6];
	PlcInputs.ST60_5_DM260_Result_Data_64_bytes[7] := HwInputs.ST60_5_DM260_Result_Data_64_bytes[7];
	PlcInputs.ST60_5_DM260_Result_Data_64_bytes[8] := HwInputs.ST60_5_DM260_Result_Data_64_bytes[8];
	PlcInputs.ST60_5_DM260_Result_Data_64_bytes[9] := HwInputs.ST60_5_DM260_Result_Data_64_bytes[9];
	PlcInputs.ST60_5_DM260_Result_Data_64_bytes[10] := HwInputs.ST60_5_DM260_Result_Data_64_bytes[10];
	PlcInputs.ST60_5_DM260_Result_Data_64_bytes[11] := HwInputs.ST60_5_DM260_Result_Data_64_bytes[11];
	PlcInputs.ST60_5_DM260_Result_Data_64_bytes[12] := HwInputs.ST60_5_DM260_Result_Data_64_bytes[12];
	PlcInputs.ST60_5_DM260_Result_Data_64_bytes[13] := HwInputs.ST60_5_DM260_Result_Data_64_bytes[13];
	PlcInputs.ST60_5_DM260_Result_Data_64_bytes[14] := HwInputs.ST60_5_DM260_Result_Data_64_bytes[14];
	PlcInputs.ST60_5_DM260_Result_Data_64_bytes[15] := HwInputs.ST60_5_DM260_Result_Data_64_bytes[15];
	PlcInputs.ST60_5_DM260_Result_Data_64_bytes[16] := HwInputs.ST60_5_DM260_Result_Data_64_bytes[16];
	PlcInputs.ST60_5_DM260_Result_Data_64_bytes[17] := HwInputs.ST60_5_DM260_Result_Data_64_bytes[17];
	PlcInputs.ST60_5_DM260_Result_Data_64_bytes[18] := HwInputs.ST60_5_DM260_Result_Data_64_bytes[18];
	PlcInputs.ST60_5_DM260_Result_Data_64_bytes[19] := HwInputs.ST60_5_DM260_Result_Data_64_bytes[19];
	PlcInputs.ST60_5_DM260_Result_Data_64_bytes[20] := HwInputs.ST60_5_DM260_Result_Data_64_bytes[20];
	PlcInputs.ST60_5_DM260_Result_Data_64_bytes[21] := HwInputs.ST60_5_DM260_Result_Data_64_bytes[21];
	PlcInputs.ST60_5_DM260_Result_Data_64_bytes[22] := HwInputs.ST60_5_DM260_Result_Data_64_bytes[22];
	PlcInputs.ST60_5_DM260_Result_Data_64_bytes[23] := HwInputs.ST60_5_DM260_Result_Data_64_bytes[23];
	PlcInputs.ST60_5_DM260_Result_Data_64_bytes[24] := HwInputs.ST60_5_DM260_Result_Data_64_bytes[24];
	PlcInputs.ST60_5_DM260_Result_Data_64_bytes[25] := HwInputs.ST60_5_DM260_Result_Data_64_bytes[25];
	PlcInputs.ST60_5_DM260_Result_Data_64_bytes[26] := HwInputs.ST60_5_DM260_Result_Data_64_bytes[26];
	PlcInputs.ST60_5_DM260_Result_Data_64_bytes[27] := HwInputs.ST60_5_DM260_Result_Data_64_bytes[27];
	PlcInputs.ST60_5_DM260_Result_Data_64_bytes[28] := HwInputs.ST60_5_DM260_Result_Data_64_bytes[28];
	PlcInputs.ST60_5_DM260_Result_Data_64_bytes[29] := HwInputs.ST60_5_DM260_Result_Data_64_bytes[29];
	PlcInputs.ST60_5_DM260_Result_Data_64_bytes[30] := HwInputs.ST60_5_DM260_Result_Data_64_bytes[30];
	PlcInputs.ST60_5_DM260_Result_Data_64_bytes[31] := HwInputs.ST60_5_DM260_Result_Data_64_bytes[31];
	PlcInputs.ST60_5_DM260_Result_Data_64_bytes[32] := HwInputs.ST60_5_DM260_Result_Data_64_bytes[32];
	PlcInputs.ST60_5_DM260_Result_Data_64_bytes[33] := HwInputs.ST60_5_DM260_Result_Data_64_bytes[33];
	PlcInputs.ST60_5_DM260_Result_Data_64_bytes[34] := HwInputs.ST60_5_DM260_Result_Data_64_bytes[34];
	PlcInputs.ST60_5_DM260_Result_Data_64_bytes[35] := HwInputs.ST60_5_DM260_Result_Data_64_bytes[35];
	PlcInputs.ST60_5_DM260_Result_Data_64_bytes[36] := HwInputs.ST60_5_DM260_Result_Data_64_bytes[36];
	PlcInputs.ST60_5_DM260_Result_Data_64_bytes[37] := HwInputs.ST60_5_DM260_Result_Data_64_bytes[37];
	PlcInputs.ST60_5_DM260_Result_Data_64_bytes[38] := HwInputs.ST60_5_DM260_Result_Data_64_bytes[38];
	PlcInputs.ST60_5_DM260_Result_Data_64_bytes[39] := HwInputs.ST60_5_DM260_Result_Data_64_bytes[39];
	PlcInputs.ST60_5_DM260_Result_Data_64_bytes[40] := HwInputs.ST60_5_DM260_Result_Data_64_bytes[40];
	PlcInputs.ST60_5_DM260_Result_Data_64_bytes[41] := HwInputs.ST60_5_DM260_Result_Data_64_bytes[41];
	PlcInputs.ST60_5_DM260_Result_Data_64_bytes[42] := HwInputs.ST60_5_DM260_Result_Data_64_bytes[42];
	PlcInputs.ST60_5_DM260_Result_Data_64_bytes[43] := HwInputs.ST60_5_DM260_Result_Data_64_bytes[43];
	PlcInputs.ST60_5_DM260_Result_Data_64_bytes[44] := HwInputs.ST60_5_DM260_Result_Data_64_bytes[44];
	PlcInputs.ST60_5_DM260_Result_Data_64_bytes[45] := HwInputs.ST60_5_DM260_Result_Data_64_bytes[45];
	PlcInputs.ST60_5_DM260_Result_Data_64_bytes[46] := HwInputs.ST60_5_DM260_Result_Data_64_bytes[46];
	PlcInputs.ST60_5_DM260_Result_Data_64_bytes[47] := HwInputs.ST60_5_DM260_Result_Data_64_bytes[47];
	PlcInputs.ST60_5_DM260_Result_Data_64_bytes[48] := HwInputs.ST60_5_DM260_Result_Data_64_bytes[48];
	PlcInputs.ST60_5_DM260_Result_Data_64_bytes[49] := HwInputs.ST60_5_DM260_Result_Data_64_bytes[49];
	PlcInputs.ST60_5_DM260_Result_Data_64_bytes[50] := HwInputs.ST60_5_DM260_Result_Data_64_bytes[50];
	PlcInputs.ST60_5_DM260_Result_Data_64_bytes[51] := HwInputs.ST60_5_DM260_Result_Data_64_bytes[51];
	PlcInputs.ST60_5_DM260_Result_Data_64_bytes[52] := HwInputs.ST60_5_DM260_Result_Data_64_bytes[52];
	PlcInputs.ST60_5_DM260_Result_Data_64_bytes[53] := HwInputs.ST60_5_DM260_Result_Data_64_bytes[53];
	PlcInputs.ST60_5_DM260_Result_Data_64_bytes[54] := HwInputs.ST60_5_DM260_Result_Data_64_bytes[54];
	PlcInputs.ST60_5_DM260_Result_Data_64_bytes[55] := HwInputs.ST60_5_DM260_Result_Data_64_bytes[55];
	PlcInputs.ST60_5_DM260_Result_Data_64_bytes[56] := HwInputs.ST60_5_DM260_Result_Data_64_bytes[56];
	PlcInputs.ST60_5_DM260_Result_Data_64_bytes[57] := HwInputs.ST60_5_DM260_Result_Data_64_bytes[57];
	PlcInputs.ST60_5_DM260_Result_Data_64_bytes[58] := HwInputs.ST60_5_DM260_Result_Data_64_bytes[58];
	PlcInputs.ST60_5_DM260_Result_Data_64_bytes[59] := HwInputs.ST60_5_DM260_Result_Data_64_bytes[59];
	PlcInputs.ST60_5_DM260_Result_Data_64_bytes[60] := HwInputs.ST60_5_DM260_Result_Data_64_bytes[60];
	PlcInputs.ST60_5_DM260_Result_Data_64_bytes[61] := HwInputs.ST60_5_DM260_Result_Data_64_bytes[61];
	PlcInputs.ST60_5_DM260_Result_Data_64_bytes[62] := HwInputs.ST60_5_DM260_Result_Data_64_bytes[62];
	PlcInputs.ST60_5_DM260_Result_Data_64_bytes[63] := HwInputs.ST60_5_DM260_Result_Data_64_bytes[63];
	PlcInputs.ST60_5_DM260_Result_Data_64_bytes[64] := HwInputs.ST60_5_DM260_Result_Data_64_bytes[64];
	PlcInputs.ST60_5_DM260_Result_Data_64_bytes[65] := HwInputs.ST60_5_DM260_Result_Data_64_bytes[65];
	PlcInputs.ST60_5_DM260_Result_Data_64_bytes[66] := HwInputs.ST60_5_DM260_Result_Data_64_bytes[66];
	PlcInputs.ST60_5_DM260_Result_Data_64_bytes[67] := HwInputs.ST60_5_DM260_Result_Data_64_bytes[67];
	PlcInputs.ST60_5_DM260_Result_Data_64_bytes[68] := HwInputs.ST60_5_DM260_Result_Data_64_bytes[68];
	PlcInputs.ST60_5_DM260_Result_Data_64_bytes[69] := HwInputs.ST60_5_DM260_Result_Data_64_bytes[69];
	PlcInputs.ST60_5_DM260_Result_Data_64_bytes[70] := HwInputs.ST60_5_DM260_Result_Data_64_bytes[70];
	PlcInputs.ST60_5_DM260_Result_Data_64_bytes[71] := HwInputs.ST60_5_DM260_Result_Data_64_bytes[71];
END_FUNCTION
